FUNCTION_BLOCK fbPPPSZadajnikSR04P
  VAR_INPUT
    sKomunikat : alSTRINGKomunikat;  (* komunikat z systemu zewnętrznego *)
    intTablicaKomunikatowRozmiar : INT;  (* rozmiar tablicy danych wysyłkowych *)
    intModbusOdczytZapisZadanieRozmiar : INT;  (* rozmiar tablicy danych modbusa *)
    xTablicaKomunikatowHold : BOOL;  (* wstrzymanie komunikacji mniej ważnych komunikatów *)
    sIdInstancji : STRING;  (* parametr ID rolety np NS02L*202IBM**** *)
    sIdAplikacji : STRING;  (* parametr ID aplikacji np SO*******ECL*000 *)
    sMnemonik : STRING;  (* mnemonik właściciela - BCB* *)
    sMACAdres : STRING;  (* MAC adres sterownika *)
    sDaneZapasowe : STRING;  (* 6 znaków zapasu *)
    tCzasOpoznieniaRestartu : TIME;  (* czas opóźnienia po którym zaczynają być raportowane wartości *)
    sTypPomieszczenia : STRING;  (* typ pomieszczenia *)
    bAdres : BYTE;
    bKanalEnOcean : BYTE;
    sEnOceanID : STRING(10);
    tMinimalnyCzasRaportowania : TIME;
    tMaksymalnyCzasRaportowania : TIME;
    tCzasTimeoutEnOcean : TIME;
    xAutonomizacja : BOOL;
    xAutonomizacjaSztuczna : BOOL;
    xGlobalnaAutomatycznaKonfiguracja : BOOL;
    tCzestotliwoscAutomatycznejKonfiguracji : TIME;
    rRegulatorTemperaturyKp : REAL;
    rRegulatorTemperaturyTi : REAL;
    rRegulatorTemperaturyDeadZone : REAL;
    rTrybPracyAutonomizacja : REAL;  (* Domyślny tryb pracy *)
    rTemperaturaBazowaAutoAutonomizacja : REAL;  (* Domyślna wartość nastawy temperatury bazowej w trybie automatycznym *)
    rTemperaturaBazowaManAutonomizacja : REAL;  (* Domyślna wartość nastawy temperatury bazowej w trybie manualnym *)
    rSkalaPotencjometruAutonomizacja : REAL;  (* Domyślna skala potencjomentru *)
    rTemperaturaBazowaHMI : REAL := 293.15;  (* Temperatura bazowa z HMI *)
    intTrybPracyHMI : INT := 1;  (* 0 - ręczny; 1 - auto *)
    xPokazPanelHMI : BOOL := TRUE;  (* 0 - widoczny; 1 - niewidoczny *)
  END_VAR
  VAR_IN_OUT
    arModbusOdczytCykliczny : ARRAY[1..5000] OF typModbusOdczytCykliczny;
    arModbusStatusKomunikacji : ARRAY[1..256] OF INT;
    arModbusOdczytZapisZadanie : ARRAY[1..1000] OF typModbusOdczytZapisZadanie;
    intModbusOdczytZapisZadanieZnacznikZapisu : INT;
    arTablicaKomunikatow : alARRAYTablicaKomunikatow;
    intTablicaKomunikatowZnacznikZapisu : INT;
  END_VAR
  VAR_OUTPUT
    rWyjscieRgulatoraTemperatury : REAL;
    rDiagnostykaTemperaturaPomieszczenia : REAL;
    rDiagnostykaTemperaturaNastawiona : REAL;
    rDiagnostykaTemperaturaBazowa : REAL;
    rDiagnostykaKorektaTemperaturyPotencjometru : REAL;
    rDiagnostykaWyjscieRgulatoraTemperatury : REAL;
    intDiagnostykaTrybPracy : INT;
    sDiagnostykaEnOceanIDodczytany : STRING(10);
    wDiagnostykaCzasOdOstatniegoKomunikatu : WORD;
    rTemperaturaPomieszczenia : REAL;
  END_VAR
  VAR CONSTANT
    uintLiczbaRejestrowNaKanal : UINT := 20;
    uintPierwszyRejestr : UINT := 200;
    wEnOceanFunction : WORD := 16;
    wEnOceanType : WORD := 3;
    wEnOceanManufacturer : WORD := 2;
    intDomyslneHarmonogram : INT := enumPPPSHarmonogramy.Komfort;  (* domyślne nastawy po restarcie sterownika *)
    rDomyslneTemperaturaBazowaKomfort : REAL := 293.15;
    rDomyslneTemperaturaBazowaEkonomiczny : REAL := 292.15;
  END_VAR
  VAR
    uintFunctionModbusAdres : UINT;  (* definicja adresów rejestrów modbusowych *)
    uintTypeModbusAdres : UINT;
    uintManufacturerModbusAdres : UINT;
    uintEnOceanIDHiModbusAdres : UINT;
    uintEnOceanIDLoModbusAdres : UINT;
    uintCzasOdOstatniegoKomunikatuModbusAdres : UINT;
    uintPustyRejestr1ModbusAdres : UINT;
    uintStatusUrzadzeniaModbusAdres : UINT;
    uintPustyRejestr2ModbusAdres : UINT;
    uintTemperaturaPomieszczeniaOdczytanaModbusAdres : UINT;
    uintNastawaPotencjometruModbusAdres : UINT;
    xPierwszySkan : BOOL := TRUE;  (* uintLiczbaTelegramowModbusAdres : UINT; zmienne operacyjne *)
    intPetlaPierwszySkan : INT := 1;
    intRozkazTymczasowy : INT;
    arNastawyRegulatoraTemperatury : typConfigPIDController;
    fbRegulatorTemperatury : FbPIDController;
    intBlokadaWykonywaniaRozkazow : INT;
    intBlokadaWykonywaniaRozkazowZaraportowana : INT;
    intTrybPracy : INT;  (* Tryb pracy regulatora. *)
    intTrybPracyZaraportowana : INT;
    xTrybPracyZapisz : BOOL;  (* Trigger zapisu wartości w pamięci urządzenia. *)
    rTrybPracyZapis : REAL;  (* Wartość do zapisania w pamięci urządzenia. *)
    rTemperaturaBazowaAuto : REAL := 293.15;  (* Temperatura bazowa trybu automatycznego. *)
    rTemperaturaBazowaAutoZaraportowana : REAL;
    xTemperaturaBazowaAutoZapisz : BOOL;  (* Trigger zapisu wartości w pamięci urządzenia. *)
    rTemperaturaBazowaAutoZapis : REAL;  (* Wartość do zapisania w pamięci urządzenia. *)
    rTemperaturaBazowaMan : REAL := 293.15;  (* Temperatura bazowa trybu manualnego. *)
    rTemperaturaBazowaManZaraportowana : REAL;
    xTemperaturaBazowaManZapisz : BOOL;  (* Trigger zapisu wartości w pamięci urządzenia. *)
    rTemperaturaBazowaManZapis : REAL;  (* Wartość do zapisania w pamięci urządzenia. *)
    rSkalaPotencjometru : REAL;  (* Skala Potencjometru *)
    rSkalaPotencjometruZaraportowana : REAL;
    xSkalaPotencjometruZapisz : BOOL;  (* Trigger zapisu wartości w pamięci urządzenia. *)
    rSkalaPotencjometruZapis : REAL;  (* Wartość do zapisania w pamięci urządzenia. *)
    fbZadanieGrzania : fbFiltrWartoscAnalogowa;
    rZadanieGrzania : REAL;  (* Zadana grzania *)
    fbZadanieGrzaniaRaport : fbFiltrWartoscAnalogowa;
    rZadanieGrzaniaRaport : REAL;  (* Zadana grzania (raportowana) *)
    rZadanieGrzaniaRaportZaraportowana : REAL;
    rWartoscWejsciowaTemperaturyNastawionej : REAL;
    fbWyslanieKonfiguracji : TON;  (* definicja zmiennych i FB do odczytu wartości z modbusa *)
    xPozwolenieNaAutomatycznaKonfiguracje : BOOL;
    xResetTimerautomatycznejKonfiguracji : BOOL;
    wFunctionEnOceanOdczytana : WORD;
    wTypeEnOceanOdczytana : WORD;
    wManufacturerEnOceanOdczytana : WORD;
    sEnOceanIDodczytany : STRING(10);
    wEnOceanIDHi : WORD;
    wEnOceanIDLo : WORD;
    wEnOceanIDHiZapis : WORD;
    wEnOceanIDLoZapis : WORD;
    wCzasOdOstatniegoKomunikatu : WORD;
    fbTimeoutEnOcean : TON;
    wStatusUrzadzenia : WORD;
    wLiczbaTelegramow : WORD;
    uintLiczbaTelegramow : UINT;
    wPustyRejestr1 : WORD;  (* Rejestry odczytywane dla zgrupowania zapytania rejestrów Modbus *)
    wPustyRejestr2 : WORD;
    wTemperaturaPomieszczeniaOdczytana : WORD;
    fbTemperaturaPomieszczenia : fbFiltrWartoscAnalogowa;
    rTemperaturaPomieszczeniaZaraportowana : REAL;
    wNastawaPotencjometru : WORD;
    rTemperaturaNastawiona : REAL;
    rTemperaturaNastawionaZaraportowana : REAL;
    xPoInicjalizacji : BOOL := FALSE;  (* inicjalizacja *)
    fbInicjalizacyjnyTimer : TON;
    sDane : alSTRINGKomunikat;
    sWyslanyKomunikat : alSTRINGKomunikat;
    sKomunikatPamiec : alSTRINGKomunikat;
    sWyslanyKomunikatDummy : alSTRINGKomunikat;
    intPetla : INT;
    arErrorStan : ARRAY[0..3] OF INT;  (* tablica przechowująca statusy alarmowe *)
    arErrorKlasa : ARRAY[0..3] OF INT;  (* tablica przechowująca klasy danych alarmów *)
    sTempWartoscAtrybutu : STRING;
    rTempWartoscAtrybutu : REAL;
    intTempWartoscAtrybutu : INT;
    xRaport : BOOL;
    uintFunctionAdres : UINT;
    sPlakietkaHMI : STRING;  (* Plakietka pomieszczenia zawierająca numer piętra i pomieszczenia (na potrzeby webvisu) *)
    fnPrzywrocDomyslne : R_TRIG;  (* Przywracanie domyślnych wartości nastaw *)
    fbTaktowanieZapisywaniaModbus : TON;  (* Cykliczne żądanie zapisu danych do urządzenia *)
    xBrakKomunikacjiEnOcean : BOOL;  (* Brak komunikacji z urządzeniem po enOcean *)
    tonBrakKomunikacjiPLC : TON;
    xBrakKomunikacjiPLC : BOOL;
    xBrakKomunikacjiIZE : BOOL;
    rTemperaturaPomieszczeniaPamiec : REAL;  (* Temperatura zapamiętana w celu porównania z aktualną *)
    xBrakZmianyTemperatury : BOOL;  (* Flaga braku zmiany temperatury *)
    fbBrakZmianyTemperaturyTimer : TON;  (* Timer braku zmiany temperatury (24 godziny) *)
    xBladBrakZmianyTemperatury : BOOL;  (* Błąd braku zmiany temperatury *)
    xOsiagniecieTemperaturyZadanej : BOOL := FALSE;  (* Sprawdzanie czy została osiągnęta zadana temperatura *)
    xOsiagniecieTemperaturyZadanejZaraportowana : BOOL := FALSE;
    xFlagaTrybuPracy : BOOL := FALSE;
    rRoznicaTemperaturyZadanejOrazZaraportowanej : REAL;
  END_VAR

            (*			
Autor:					Paweł Kąkol, 2018-08-06, Artur Wyszomirski
Prawa majątkowe: 		Solwena Sp. z o.o., 
Aktualizacje:			
						2018-08-27-PK: dodanie algorytmu nadpisywania konfiguracji (uczenia) anteny
						2018-09-10-PK: dodanie regulatora temperatury oraz obsługi atrybutów potrzebnych do zadajnika z regulatorem, dodanie alarmowania Timeout komunikacji EnOcean
						2018-09-24-AWy: obsługa trybu manualnego i automatycznego
						2018-09-25-PK: dodanie domyślnego przyjmowania 21 st. C po restarcie sterownika, zanim nastąpi Autonomizacja i komunikacja z IZE.
						2018-15-10-AWy: obsługa harmonogramów
						2018-23-10-JB: przygotowanie atrybutów i alarmów do komunikacji z IZE
						2018-12-12-JB: napisanie od nowa obsługi ramek typu C i Q
						2019-02-26-JB: zmiana deadbandów w filtrach analogowych
						2019-04-08-AWy: usunięcie buga braku wysterowania grzejników w trybie manualnym (usunięcie intTrybPracy <> enumPPPSZadajnikTrybPracy.Manualny AND z linii 473)
						2019-05-13-AWy: zmiana wartości umieszczonej w atrybucie STERGRZ. Wartość rZadanieGrzania jest dzielona przez 100 tak, aby zakres STERGRZ mieścił się między 0 a 1.
						2019-05-16-AWy: modyfikacja warunku na raportowanie. Dopisane: AND arModbusStatusKomunikacji[bAdres] = enumModbusStatus.KomunikacjaPrawidlowa AND xPoInicjalizacji 
						2019-05-17-AWy: rozbicie zmiennej rTemperaturaBazowa na rTemperaturaBazowaAuto i rTemperaturaBazowaMan
						2019-05-21-AWy: modyfikacja przepisywania temperatury bazowej z IZE do lokalnej podczas regulacji IZE. 
						2019-06-05-AWy: załadowanie domyślnych trybów pracy i nastaw po przejściu w tryb autonomizacji
						2019-08-05-AWy: dodanie zmiennej sPlakietkaHMI.
						2019-08-14-AWy: zmiana fbPrzywrocDomyslne z przerzutnika RS na R_TRIG.
						2019-09-23-AWy: modyfikacja generowania wartości zmiennej xBrakKomunikacjiPLC
						2019-10-09-AWy: uzależnienie wystąpienia alarmu braku zmiany temperatury od stanu komunikacji 
						2019-10-10-AWy: przywrócenie zmiennej xBrakKomunikacjiEnOcean na potrzeby alarmów i webvisu z I etapu ENGIE
						2019-10-21-AWy: dodanie dodatkowego filtrowania zadanej grzania przy wysyłaniu ramek do IZE
						2019-10-22-AWy: usunięcie uintLiczbaTelegramowModbusAdres z odczytu po Modbusie
						
Opis:					fb służy do komunikacji po Modbus RTU za pośrednictwem bramek (STC65-RS485) EnOcean z zadajnikami FCP0 (SR04P) na budynkach PPP Sopot (ENGIE) 
*)

// Inicjalizacja sterownika
fbInicjalizacyjnyTimer(IN := NOT xPoInicjalizacji , PT := tCzasOpoznieniaRestartu);
IF fbInicjalizacyjnyTimer.Q THEN
	intTrybPracyZaraportowana := intTrybPracy;
	rTemperaturaBazowaAutoZaraportowana := rTemperaturaBazowaAuto;
	rTemperaturaBazowaManZaraportowana := rTemperaturaBazowaMan;
	rSkalaPotencjometruZaraportowana := rSkalaPotencjometru;
	rTemperaturaNastawionaZaraportowana := rTemperaturaNastawiona;
	rTemperaturaPomieszczeniaZaraportowana := rTemperaturaPomieszczenia;
	rZadanieGrzaniaRaportZaraportowana := rZadanieGrzaniaRaport;
	xOsiagniecieTemperaturyZadanej := xOsiagniecieTemperaturyZadanejZaraportowana;
	xPoInicjalizacji := TRUE;
END_IF

// Włącz autonomizację jeśli sterownik jest w stanie inicjalizacji lub nastąpiło wymuszenie autonomizacji
IF NOT xPoInicjalizacji OR xAutonomizacjaSztuczna = TRUE THEN
	xAutonomizacja := TRUE;
END_IF 

// Kontrola komunikacji
tonBrakKomunikacjiPLC(IN := (wCzasOdOstatniegoKomunikatu > 180 OR arModbusStatusKomunikacji[bAdres] <> enumModbusStatus.KomunikacjaPrawidlowa), PT := T#180S);
IF tonBrakKomunikacjiPLC.Q THEN
	xBrakKomunikacjiPLC := TRUE;
ELSE
	xBrakKomunikacjiPLC := FALSE;
END_IF

IF xAutonomizacja THEN
	xBrakKomunikacjiIZE := TRUE;
ELSE
	xBrakKomunikacjiIZE := FALSE;
END_IF

IF xPierwszySkan THEN
	xPierwszySkan := FALSE;
	WHILE arModbusOdczytCykliczny[intPetlaPierwszySkan].bAdresUrzadzenia <> 0 DO
		intPetlaPierwszySkan := intPetlaPierwszySkan + 1;
	END_WHILE
	
	//ustawienie parametrów regulatora temperatury
	arNastawyRegulatoraTemperatury.rKp := rRegulatorTemperaturyKp;
	arNastawyRegulatoraTemperatury.rTn := rRegulatorTemperaturyTi;
	arNastawyRegulatoraTemperatury.rTd := 0.0;
	arNastawyRegulatoraTemperatury.rOutputMax := 100.0;
	arNastawyRegulatoraTemperatury.rOutputMin := 0.0;
	arNastawyRegulatoraTemperatury.xPresetOn := TRUE;
	arNastawyRegulatoraTemperatury.rPresetValueOn := 0.0;
	arNastawyRegulatoraTemperatury.rPresetValueOff := 0.0;
	arNastawyRegulatoraTemperatury.rDeadZone := rRegulatorTemperaturyDeadZone;
	
	//wyznaczenie adresów rejestrów modbusowych
	uintFunctionModbusAdres := uintPierwszyRejestr + (uintLiczbaRejestrowNaKanal * (BYTE_TO_UINT(bKanalEnOcean) - 1));
	uintTypeModbusAdres := uintFunctionModbusAdres + 1;
	uintManufacturerModbusAdres := uintFunctionModbusAdres + 2;
	
	uintEnOceanIDHiModbusAdres := uintFunctionModbusAdres + 3;
	uintEnOceanIDLoModbusAdres := uintFunctionModbusAdres + 4;
	uintCzasOdOstatniegoKomunikatuModbusAdres := uintFunctionModbusAdres + 6;
	uintPustyRejestr1ModbusAdres := uintFunctionModbusAdres + 7;
	uintStatusUrzadzeniaModbusAdres := uintFunctionModbusAdres + 8;
	uintPustyRejestr2ModbusAdres := uintFunctionModbusAdres + 9;
	uintTemperaturaPomieszczeniaOdczytanaModbusAdres := uintFunctionModbusAdres + 10;
	uintNastawaPotencjometruModbusAdres := uintFunctionModbusAdres + 11;
	//uintLiczbaTelegramowModbusAdres := uintFunctionModbusAdres + 19;
	
//deklaracja rejestrow do odczytu
	//rejestry
	arModbusOdczytCykliczny[intPetlaPierwszySkan].bAdresUrzadzenia := bAdres;
	arModbusOdczytCykliczny[intPetlaPierwszySkan].bFunkcja := TO_BYTE(enumModbusKodyFunkcji.OdczytNRejestrow);
	arModbusOdczytCykliczny[intPetlaPierwszySkan].uiAdresRejestru := uintFunctionModbusAdres;
	arModbusOdczytCykliczny[intPetlaPierwszySkan].ltCzestotliwosc := TIME_TO_LTIME(tMaksymalnyCzasRaportowania);
	arModbusOdczytCykliczny[intPetlaPierwszySkan].pZmiennaReferencyjna := ADR(wFunctionEnOceanOdczytana);
	intPetlaPierwszySkan := intPetlaPierwszySkan + 1;
	
	arModbusOdczytCykliczny[intPetlaPierwszySkan].bAdresUrzadzenia := bAdres;
	arModbusOdczytCykliczny[intPetlaPierwszySkan].bFunkcja := TO_BYTE(enumModbusKodyFunkcji.OdczytNRejestrow);
	arModbusOdczytCykliczny[intPetlaPierwszySkan].uiAdresRejestru := uintTypeModbusAdres;
	arModbusOdczytCykliczny[intPetlaPierwszySkan].ltCzestotliwosc := TIME_TO_LTIME(tMaksymalnyCzasRaportowania);
	arModbusOdczytCykliczny[intPetlaPierwszySkan].pZmiennaReferencyjna := ADR(wTypeEnOceanOdczytana);
	intPetlaPierwszySkan := intPetlaPierwszySkan + 1;
	
	arModbusOdczytCykliczny[intPetlaPierwszySkan].bAdresUrzadzenia := bAdres;
	arModbusOdczytCykliczny[intPetlaPierwszySkan].bFunkcja := TO_BYTE(enumModbusKodyFunkcji.OdczytNRejestrow);
	arModbusOdczytCykliczny[intPetlaPierwszySkan].uiAdresRejestru := uintManufacturerModbusAdres;
	arModbusOdczytCykliczny[intPetlaPierwszySkan].ltCzestotliwosc := TIME_TO_LTIME(tMaksymalnyCzasRaportowania);
	arModbusOdczytCykliczny[intPetlaPierwszySkan].pZmiennaReferencyjna := ADR(wManufacturerEnOceanOdczytana);
	intPetlaPierwszySkan := intPetlaPierwszySkan + 1;
	
	arModbusOdczytCykliczny[intPetlaPierwszySkan].bAdresUrzadzenia := bAdres;
	arModbusOdczytCykliczny[intPetlaPierwszySkan].bFunkcja := TO_BYTE(enumModbusKodyFunkcji.OdczytNRejestrow);
	arModbusOdczytCykliczny[intPetlaPierwszySkan].uiAdresRejestru := uintEnOceanIDHiModbusAdres;
	arModbusOdczytCykliczny[intPetlaPierwszySkan].ltCzestotliwosc := TIME_TO_LTIME(tMaksymalnyCzasRaportowania);
	arModbusOdczytCykliczny[intPetlaPierwszySkan].pZmiennaReferencyjna := ADR(wEnOceanIDHi);
	intPetlaPierwszySkan := intPetlaPierwszySkan + 1;
	
	arModbusOdczytCykliczny[intPetlaPierwszySkan].bAdresUrzadzenia := bAdres;
	arModbusOdczytCykliczny[intPetlaPierwszySkan].bFunkcja := TO_BYTE(enumModbusKodyFunkcji.OdczytNRejestrow);
	arModbusOdczytCykliczny[intPetlaPierwszySkan].uiAdresRejestru := uintEnOceanIDLoModbusAdres;
	arModbusOdczytCykliczny[intPetlaPierwszySkan].ltCzestotliwosc := TIME_TO_LTIME(tMaksymalnyCzasRaportowania);
	arModbusOdczytCykliczny[intPetlaPierwszySkan].pZmiennaReferencyjna := ADR(wEnOceanIDLo);
	intPetlaPierwszySkan := intPetlaPierwszySkan + 1;
	
	arModbusOdczytCykliczny[intPetlaPierwszySkan].bAdresUrzadzenia := bAdres;
	arModbusOdczytCykliczny[intPetlaPierwszySkan].bFunkcja := TO_BYTE(enumModbusKodyFunkcji.OdczytNRejestrow);
	arModbusOdczytCykliczny[intPetlaPierwszySkan].uiAdresRejestru := uintCzasOdOstatniegoKomunikatuModbusAdres;
	arModbusOdczytCykliczny[intPetlaPierwszySkan].ltCzestotliwosc := TIME_TO_LTIME(tMinimalnyCzasRaportowania);
	arModbusOdczytCykliczny[intPetlaPierwszySkan].pZmiennaReferencyjna := ADR(wCzasOdOstatniegoKomunikatu);
	intPetlaPierwszySkan := intPetlaPierwszySkan + 1;
	
	arModbusOdczytCykliczny[intPetlaPierwszySkan].bAdresUrzadzenia := bAdres;
	arModbusOdczytCykliczny[intPetlaPierwszySkan].bFunkcja := TO_BYTE(enumModbusKodyFunkcji.OdczytNRejestrow);
	arModbusOdczytCykliczny[intPetlaPierwszySkan].uiAdresRejestru := uintPustyRejestr1ModbusAdres;
	arModbusOdczytCykliczny[intPetlaPierwszySkan].ltCzestotliwosc := TIME_TO_LTIME(tMinimalnyCzasRaportowania);
	arModbusOdczytCykliczny[intPetlaPierwszySkan].pZmiennaReferencyjna := ADR(wPustyRejestr1);
	intPetlaPierwszySkan := intPetlaPierwszySkan + 1;
	
	arModbusOdczytCykliczny[intPetlaPierwszySkan].bAdresUrzadzenia := bAdres;
	arModbusOdczytCykliczny[intPetlaPierwszySkan].bFunkcja := TO_BYTE(enumModbusKodyFunkcji.OdczytNRejestrow);
	arModbusOdczytCykliczny[intPetlaPierwszySkan].uiAdresRejestru := uintStatusUrzadzeniaModbusAdres;
	arModbusOdczytCykliczny[intPetlaPierwszySkan].ltCzestotliwosc := TIME_TO_LTIME(tMinimalnyCzasRaportowania);
	arModbusOdczytCykliczny[intPetlaPierwszySkan].pZmiennaReferencyjna := ADR(wStatusUrzadzenia);
	intPetlaPierwszySkan := intPetlaPierwszySkan + 1;
	
	arModbusOdczytCykliczny[intPetlaPierwszySkan].bAdresUrzadzenia := bAdres;
	arModbusOdczytCykliczny[intPetlaPierwszySkan].bFunkcja := TO_BYTE(enumModbusKodyFunkcji.OdczytNRejestrow);
	arModbusOdczytCykliczny[intPetlaPierwszySkan].uiAdresRejestru := uintPustyRejestr2ModbusAdres;
	arModbusOdczytCykliczny[intPetlaPierwszySkan].ltCzestotliwosc := TIME_TO_LTIME(tMinimalnyCzasRaportowania);
	arModbusOdczytCykliczny[intPetlaPierwszySkan].pZmiennaReferencyjna := ADR(wPustyRejestr2);
	intPetlaPierwszySkan := intPetlaPierwszySkan + 1;
	
	arModbusOdczytCykliczny[intPetlaPierwszySkan].bAdresUrzadzenia := bAdres;
	arModbusOdczytCykliczny[intPetlaPierwszySkan].bFunkcja := TO_BYTE(enumModbusKodyFunkcji.OdczytNRejestrow);
	arModbusOdczytCykliczny[intPetlaPierwszySkan].uiAdresRejestru := uintTemperaturaPomieszczeniaOdczytanaModbusAdres;
	arModbusOdczytCykliczny[intPetlaPierwszySkan].ltCzestotliwosc := TIME_TO_LTIME(tMinimalnyCzasRaportowania);
	arModbusOdczytCykliczny[intPetlaPierwszySkan].pZmiennaReferencyjna := ADR(wTemperaturaPomieszczeniaOdczytana);
	intPetlaPierwszySkan := intPetlaPierwszySkan + 1;	
	
	arModbusOdczytCykliczny[intPetlaPierwszySkan].bAdresUrzadzenia := bAdres;
	arModbusOdczytCykliczny[intPetlaPierwszySkan].bFunkcja := TO_BYTE(enumModbusKodyFunkcji.OdczytNRejestrow);
	arModbusOdczytCykliczny[intPetlaPierwszySkan].uiAdresRejestru := uintNastawaPotencjometruModbusAdres;
	arModbusOdczytCykliczny[intPetlaPierwszySkan].ltCzestotliwosc := TIME_TO_LTIME(tMinimalnyCzasRaportowania);
	arModbusOdczytCykliczny[intPetlaPierwszySkan].pZmiennaReferencyjna := ADR(wNastawaPotencjometru);
	intPetlaPierwszySkan := intPetlaPierwszySkan + 1;
(*	
	arModbusOdczytCykliczny[intPetlaPierwszySkan].bAdresUrzadzenia := bAdres;
	arModbusOdczytCykliczny[intPetlaPierwszySkan].bFunkcja := TO_BYTE(enumModbusKodyFunkcji.OdczytNRejestrow);
	arModbusOdczytCykliczny[intPetlaPierwszySkan].uiAdresRejestru := uintLiczbaTelegramowModbusAdres;
	arModbusOdczytCykliczny[intPetlaPierwszySkan].ltCzestotliwosc := TIME_TO_LTIME(tMinimalnyCzasRaportowania);
	arModbusOdczytCykliczny[intPetlaPierwszySkan].pZmiennaReferencyjna := ADR(wLiczbaTelegramow);
	intPetlaPierwszySkan := intPetlaPierwszySkan + 1;
*)	
(*	//przyjęcie nastaw domyślnych do momentu uzyskania nastaw z IZE lub przejścia w autonomizację
	IF intDomyslneHarmonogram = enumPPPSHarmonogramy.Ekonomiczny THEN
		rTemperaturaBazowaAuto := rDomyslneTemperaturaBazowaEkonomiczny;
	ELSE
		rTemperaturaBazowaAuto := rDomyslneTemperaturaBazowaKomfort;													
	END_IF
	intTrybPracy := enumPPPSZadajnikTrybPracy.Automatyczny;
	rSkalaPotencjometru := rSkalaPotencjometruAutonomizacja;	*)
END_IF

// Obsługa komunikatu przychodzacego z IZE
IF 	sKomunikat <> sKomunikatPamiec AND xPoInicjalizacji THEN
	sKomunikatPamiec := sKomunikat;
	IF fnIDOdbiorcyMatch(sKomunikat , sIdInstancji) THEN
		sDane := '';
		// Rozkaz typu C
		IF fnKomunikatTyp(sKomunikat) = 'C' AND NOT xAutonomizacja THEN
			// Blokada wykonywania rozkazów
			IF fnKomunikatDaneSzukajWartosci(sKomunikat,'BLOK=') = '0' THEN
				IF intBlokadaWykonywaniaRozkazow = 1 THEN
					intBlokadaWykonywaniaRozkazow := 0;
					xRaport := TRUE;
					ELSE	
					IF sDane <> '' THEN
					sDane := CONCAT(sDane , ';');
					END_IF
					sDane := CONCAT(sDane , 'BLOK=0');
				END_IF
			END_IF
			IF fnKomunikatDaneSzukajWartosci(sKomunikat,'BLOK=') = '1' THEN
				IF intBlokadaWykonywaniaRozkazow = 0 THEN
					intBlokadaWykonywaniaRozkazow := 1;
					xRaport := TRUE;
					ELSE
					IF sDane <> '' THEN
					sDane := CONCAT(sDane , ';');
					END_IF					
					sDane := CONCAT(sDane , 'BLOK=1');
				END_IF
			END_IF		

			IF intBlokadaWykonywaniaRozkazow = 0 THEN
				// Tryby pracy 
				fnKomunikatDaneZnajdzPorownajZapisz(sKomunikat := sKomunikat,
					sAtrybut := 'TRYB=',
					rAtrybutWartosc := rTrybPracyZapis,
					sDane := sDane,
					xAtrybutZapisz => xTrybPracyZapisz);	
				// Temperatura bazowa w trybie automatycznym
				fnKomunikatDaneZnajdzPorownajZapisz(sKomunikat := sKomunikat,
					sAtrybut := 'TEMPBAZAUTO=',
					rAtrybutWartosc := rTemperaturaBazowaAutoZapis,
					sDane := sDane,
					xAtrybutZapisz => xTemperaturaBazowaAutoZapisz);	
				// Temperatura bazowa w trybie manualnym
				fnKomunikatDaneZnajdzPorownajZapisz(sKomunikat := sKomunikat,
					sAtrybut := 'TEMPBAZMAN=',
					rAtrybutWartosc := rTemperaturaBazowaManZapis,
					sDane := sDane,
					xAtrybutZapisz => xTemperaturaBazowaManZapisz);
				// Skala potencjometru
				fnKomunikatDaneZnajdzPorownajZapisz(sKomunikat := sKomunikat,
					sAtrybut := 'SKALAPOT=',
					rAtrybutWartosc := rSkalaPotencjometruZapis,
					sDane := sDane,
					xAtrybutZapisz => xSkalaPotencjometruZapisz);
			END_IF
		END_IF	

		// Zapytanie typu Q
		IF fnKomunikatTyp(sKomunikat) = 'Q' AND arModbusStatusKomunikacji[bAdres] = enumModbusStatus.KomunikacjaPrawidlowa THEN
			IF fnKomunikatDaneSzukajWartosci(sKomunikat , 'BLOK=') = '?' OR fnKomunikatDaneSzukajWartosci(sKomunikat , 'ALL=') = '?' THEN
				fnKomunikatDaneDodaj(sDane := sDane , sAtrybut := 'BLOK=' , sWartosc := INT_TO_STRING(intBlokadaWykonywaniaRozkazow));	
			END_IF
			IF fnKomunikatDaneSzukajWartosci(sKomunikat , 'TRYB=') = '?' OR fnKomunikatDaneSzukajWartosci(sKomunikat , 'ALL=') = '?' THEN
				fnKomunikatDaneDodaj(sDane := sDane , sAtrybut := 'TRYB=' , sWartosc := INT_TO_STRING(intTrybPracy));	
			END_IF
			IF (fnKomunikatDaneSzukajWartosci(sKomunikat , 'TEMPBAZMAN=') = '?' OR fnKomunikatDaneSzukajWartosci(sKomunikat , 'ALL=') = '?') THEN
				fnKomunikatDaneDodaj(sDane := sDane , sAtrybut := 'TEMPBAZMAN=' , sWartosc := REAL_TO_STRING(rTemperaturaBazowaMan));	
			END_IF
			IF (fnKomunikatDaneSzukajWartosci(sKomunikat , 'TEMPBAZAUTO=') = '?' OR fnKomunikatDaneSzukajWartosci(sKomunikat , 'ALL=') = '?') THEN
				fnKomunikatDaneDodaj(sDane := sDane , sAtrybut := 'TEMPBAZAUTO=' , sWartosc := REAL_TO_STRING(rTemperaturaBazowaAuto));	
			END_IF
			IF fnKomunikatDaneSzukajWartosci(sKomunikat , 'SKALAPOT=') = '?' OR fnKomunikatDaneSzukajWartosci(sKomunikat , 'ALL=') = '?' THEN
				fnKomunikatDaneDodaj(sDane := sDane , sAtrybut := 'SKALAPOT=' , sWartosc := REAL_TO_STRING(rSkalaPotencjometru));	
			END_IF
			IF fnKomunikatDaneSzukajWartosci(sKomunikat , 'TEMP=') = '?' OR fnKomunikatDaneSzukajWartosci(sKomunikat , 'ALL=') = '?' THEN
				fnKomunikatDaneDodaj(sDane := sDane , sAtrybut := 'TEMP=' , sWartosc := REAL_TO_STRING(rTemperaturaPomieszczenia));	
			END_IF
			IF fnKomunikatDaneSzukajWartosci(sKomunikat , 'STERGRZ=') = '?' OR fnKomunikatDaneSzukajWartosci(sKomunikat , 'ALL=') = '?' THEN
				fnKomunikatDaneDodaj(sDane := sDane , sAtrybut := 'STERGRZ=' , sWartosc := REAL_TO_STRING(rZadanieGrzaniaRaport / 100));	
			END_IF
			IF fnKomunikatDaneSzukajWartosci(sKomunikat , 'TEMPNAS=') = '?' OR fnKomunikatDaneSzukajWartosci(sKomunikat , 'ALL=') = '?' THEN
				fnKomunikatDaneDodaj(sDane := sDane , sAtrybut := 'TEMPNAS=' , sWartosc := REAL_TO_STRING(rTemperaturaNastawiona));	
			END_IF
			IF fnKomunikatDaneSzukajWartosci(sKomunikat , 'DOGRZ=') = '?' OR fnKomunikatDaneSzukajWartosci(sKomunikat , 'ALL=') = '?' THEN
				fnKomunikatDaneDodaj(sDane := sDane , sAtrybut := 'DOGRZ=' , sWartosc := INT_TO_STRING(BOOL_TO_INT(xOsiagniecieTemperaturyZadanej)));	
			END_IF
			//pytanie o stany alarmów
			IF fnKomunikatDaneSzukajWartosci(sKomunikat , 'ALARM=') = '?' OR fnKomunikatDaneSzukajWartosci(sKomunikat , 'ALL=') = '?' THEN
				FOR intPetla := 1 TO 4 BY 1 DO
					//raportowanie typu E (stanów alarmów) na zapytanie typu Q
					IF arErrorStan[intPetla] <> enumAlarmWartosc.StanNieznany THEN
						fnZapiszKomunikat(	sCalyKomunikat := '' ,
											sTypKomunikatu := 'E' ,
											sMnemonik := sMnemonik ,
											sMACAdres := sMACAdres ,
											sIDNadawcy := sIdInstancji ,
											sIDOdbiorcy := sIdAplikacji ,
											sDaneZapasowe := sDaneZapasowe ,
											sDane := fnKomunikatDaneErrorRetry(xAktywny := arErrorStan[intPetla] = enumAlarmWartosc.StanAlarmowy , intKlasa := arErrorKlasa[intPetla] , intNumer := intPetla),
											arTablicaKomunikatow := arTablicaKomunikatow ,
											intTablicaKomunikatowZnacznikZapisu := intTablicaKomunikatowZnacznikZapisu ,
											intTablicaKomunikatowRozmiar := intTablicaKomunikatowRozmiar ,
											sWyslanyKomunikat := sWyslanyKomunikatDummy);
					END_IF
				END_FOR
			END_IF
		END_IF
		
		// Raportowanie typu A
		IF sDane <> '' THEN
			fnZapiszKomunikat(	sCalyKomunikat := '' ,
								sTypKomunikatu := 'A' ,
								sMnemonik := sMnemonik ,
								sMACAdres := sMACAdres ,
								sIDNadawcy := sIdInstancji ,
								sIDOdbiorcy := sIdAplikacji ,
								sDaneZapasowe := sDaneZapasowe ,
								sDane := sDane ,
								arTablicaKomunikatow := arTablicaKomunikatow ,
								intTablicaKomunikatowZnacznikZapisu := intTablicaKomunikatowZnacznikZapisu ,
								intTablicaKomunikatowRozmiar := intTablicaKomunikatowRozmiar ,
								sWyslanyKomunikat := sWyslanyKomunikatDummy);
		END_IF
	END_IF
END_IF

// Przywrócenie wartości domyślnych nastaw krzywej grzewczej i trybów pracy w przypadku restartu sterownika lub przejścia w stan autonomizacji (brak komunikacji z IZE)
fnPrzywrocDomyslne(CLK := xAutonomizacja);
IF fnPrzywrocDomyslne.Q THEN	
	IF intTrybPracy <> REAL_TO_INT(rTrybPracyAutonomizacja) THEN
		rTrybPracyZapis := rTrybPracyAutonomizacja;
		xTrybPracyZapisz := TRUE;
	END_IF
	IF rTemperaturaBazowaAuto <> rTemperaturaBazowaAutoAutonomizacja THEN
		rTemperaturaBazowaAutoZapis := rTemperaturaBazowaAutoAutonomizacja + 273.15;
		xTemperaturaBazowaAutoZapisz := TRUE;
	END_IF
	IF rTemperaturaBazowaMan <> rTemperaturaBazowaManAutonomizacja THEN
		rTemperaturaBazowaManZapis := rTemperaturaBazowaManAutonomizacja;
		xTemperaturaBazowaManZapisz := TRUE;
	END_IF
	IF rSkalaPotencjometru <> rSkalaPotencjometruAutonomizacja THEN
		rSkalaPotencjometruZapis := rSkalaPotencjometruAutonomizacja;
		xSkalaPotencjometruZapisz := TRUE;
	END_IF
END_IF	

// Zapisanie nastaw domyślnych lub otrzymanych w ramce C
IF xTrybPracyZapisz THEN
	intTrybPracy := REAL_TO_INT(rTrybPracyZapis);
	intTrybPracyHMI := REAL_TO_INT(rTrybPracyZapis);
	xTrybPracyZapisz := FALSE;
END_IF
IF xTemperaturaBazowaAutoZapisz THEN
	rTemperaturaBazowaAuto := rTemperaturaBazowaAutoZapis;
	xTemperaturaBazowaAutoZapisz := FALSE;
END_IF
IF xTemperaturaBazowaManZapisz THEN
	rTemperaturaBazowaMan := rTemperaturaBazowaManZapis;
	xTemperaturaBazowaManZapisz := FALSE;
END_IF
IF xSkalaPotencjometruZapisz THEN
	rSkalaPotencjometru := rSkalaPotencjometruZapis;
	xSkalaPotencjometruZapisz := FALSE;
END_IF

// Tryby pracy
IF xAutonomizacja THEN	// W trybie automonizacji pobieraj tryb pracy i temperaturę bazową z panelu WebVisu
	IF intTrybPracyHMI = enumPPPSZadajnikTrybPracy.Manualny THEN	
		intTrybPracy := enumPPPSZadajnikTrybPracy.Manualny;
		rTemperaturaBazowaMan := rTemperaturaBazowaHMI + 273.15;
	ELSE
		intTrybPracy := enumPPPSZadajnikTrybPracy.Automatyczny;
		rTemperaturaBazowaAuto := rTemperaturaBazowaAutoAutonomizacja + 273.15;
	END_IF
ELSE // W trybie sterowania z IZE pobieraj tryb pracy i temperaturę bazową z panelu WebVisu
	IF intTrybPracy = enumPPPSZadajnikTrybPracy.Manualny THEN
		intTrybPracyHMI := enumPPPSZadajnikTrybPracy.Manualny;
		rTemperaturaBazowaHMI := rTemperaturaBazowaMan - 273.15;
	ELSE
		intTrybPracyHMI := enumPPPSZadajnikTrybPracy.Automatyczny;
		rTemperaturaBazowaHMI := rTemperaturaBazowaAuto - 273.15;
	END_IF	
END_IF
						 
IF intTrybPracy = enumPPPSZadajnikTrybPracy.Manualny THEN 	
	rTemperaturaNastawiona := rTemperaturaBazowaMan; // W trybie manualnym nie uwzględniaj nastawy potencjometru na zadajniku
ELSE
	rTemperaturaNastawiona := ((WORD_TO_REAL(wNastawaPotencjometru) - 127.0) * rSkalaPotencjometru / 127.0) + rTemperaturaBazowaAuto; // W trybie automatycznym uwzględnij nastawę Potencjometru
END_IF

//Autokonfiguracja bramki EnOcean
sEnOceanIDodczytany := CONCAT(CONCAT(fnKonwersjaDEC_BYTE_TO_HEX_STRING(INT_TO_BYTE(WORD_TO_INT(wEnOceanIDHi / 256))), fnKonwersjaDEC_BYTE_TO_HEX_STRING(WORD_TO_BYTE(wEnOceanIDHi))), CONCAT(fnKonwersjaDEC_BYTE_TO_HEX_STRING(INT_TO_BYTE(WORD_TO_INT(wEnOceanIDLo / 256))), fnKonwersjaDEC_BYTE_TO_HEX_STRING(WORD_TO_BYTE(wEnOceanIDLo))));

fbWyslanieKonfiguracji(IN := ((xPozwolenieNaAutomatycznaKonfiguracje OR xGlobalnaAutomatycznaKonfiguracja) AND NOT xResetTimerautomatycznejKonfiguracji) , PT := tCzestotliwoscAutomatycznejKonfiguracji);
xResetTimerautomatycznejKonfiguracji := FALSE;

IF((xPozwolenieNaAutomatycznaKonfiguracje OR xGlobalnaAutomatycznaKonfiguracja) AND fbWyslanieKonfiguracji.Q) THEN
	//EnOcean ID urządzenia
	IF sEnOceanID <> sEnOceanIDodczytany THEN
		wEnOceanIDHiZapis := BYTE_TO_WORD(fnKonwersjaHEX_STRING_TO_DEC_BYTE(LEFT(sEnOceanID, 2))) * 256 + BYTE_TO_WORD(fnKonwersjaHEX_STRING_TO_DEC_BYTE(LEFT(RIGHT(sEnOceanID, 6), 2)));
		fnModbusZapisRejestru(	bAdresUrzadzenia := bAdres,
								bFunkcja := INT_TO_BYTE(enumModbusKodyFunkcji.ZapisRejestru),										
								uiAdresRejestru := uintEnOceanIDHiModbusAdres,
								pZmiennaReferencyjna := 0,
								wWartoscDoZapisania := wEnOceanIDHiZapis,
								intModbusOdczytZapisZadanieRozmiar := intModbusOdczytZapisZadanieRozmiar,
								arModbusOdczytZapisZadanie := arModbusOdczytZapisZadanie,
								intModbusOdczytZapisZadanieZnacznikZapisu := intModbusOdczytZapisZadanieZnacznikZapisu);
		wEnOceanIDLoZapis := BYTE_TO_WORD(fnKonwersjaHEX_STRING_TO_DEC_BYTE(LEFT(RIGHT(sEnOceanID, 4), 2))) * 256 + BYTE_TO_WORD(fnKonwersjaHEX_STRING_TO_DEC_BYTE(RIGHT(sEnOceanID, 2)));
		fnModbusZapisRejestru(	bAdresUrzadzenia := bAdres,
								bFunkcja := INT_TO_BYTE(enumModbusKodyFunkcji.ZapisRejestru),										
								uiAdresRejestru := uintEnOceanIDLoModbusAdres,
								pZmiennaReferencyjna := 0,
								wWartoscDoZapisania := wEnOceanIDLoZapis,
								intModbusOdczytZapisZadanieRozmiar := intModbusOdczytZapisZadanieRozmiar,
								arModbusOdczytZapisZadanie := arModbusOdczytZapisZadanie,
								intModbusOdczytZapisZadanieZnacznikZapisu := intModbusOdczytZapisZadanieZnacznikZapisu);
	END_IF
	//stałe wartości dla danego typu urządzeń
	IF wFunctionEnOceanOdczytana <> wEnOceanFunction THEN
		fnModbusZapisRejestru(	bAdresUrzadzenia := bAdres,
								bFunkcja := INT_TO_BYTE(enumModbusKodyFunkcji.ZapisRejestru),										
								uiAdresRejestru := uintFunctionModbusAdres,
								pZmiennaReferencyjna := 0,
								wWartoscDoZapisania := wEnOceanFunction,
								intModbusOdczytZapisZadanieRozmiar := intModbusOdczytZapisZadanieRozmiar,
								arModbusOdczytZapisZadanie := arModbusOdczytZapisZadanie,
								intModbusOdczytZapisZadanieZnacznikZapisu := intModbusOdczytZapisZadanieZnacznikZapisu);
	END_IF
	IF wTypeEnOceanOdczytana <> wEnOceanType THEN
		fnModbusZapisRejestru(	bAdresUrzadzenia := bAdres,
								bFunkcja := INT_TO_BYTE(enumModbusKodyFunkcji.ZapisRejestru),										
								uiAdresRejestru := uintTypeModbusAdres,
								pZmiennaReferencyjna := 0,
								wWartoscDoZapisania := wEnOceanType,
								intModbusOdczytZapisZadanieRozmiar := intModbusOdczytZapisZadanieRozmiar,
								arModbusOdczytZapisZadanie := arModbusOdczytZapisZadanie,
								intModbusOdczytZapisZadanieZnacznikZapisu := intModbusOdczytZapisZadanieZnacznikZapisu);
	END_IF
	IF wManufacturerEnOceanOdczytana <> wEnOceanManufacturer THEN
		fnModbusZapisRejestru(	bAdresUrzadzenia := bAdres,
								bFunkcja := INT_TO_BYTE(enumModbusKodyFunkcji.ZapisRejestru),										
								uiAdresRejestru := uintManufacturerModbusAdres,
								pZmiennaReferencyjna := 0,
								wWartoscDoZapisania := wEnOceanManufacturer,
								intModbusOdczytZapisZadanieRozmiar := intModbusOdczytZapisZadanieRozmiar,
								arModbusOdczytZapisZadanie := arModbusOdczytZapisZadanie,
								intModbusOdczytZapisZadanieZnacznikZapisu := intModbusOdczytZapisZadanieZnacznikZapisu);
	END_IF
	xResetTimerautomatycznejKonfiguracji := TRUE;
END_IF

//sprawdzanie Timeout komunikacji
fbTimeoutEnOcean(IN := ((wCzasOdOstatniegoKomunikatu > 120) AND arModbusStatusKomunikacji[bAdres] = enumModbusStatus.KomunikacjaPrawidlowa) , PT := tCzasTimeoutEnOcean);	
							
fbTemperaturaPomieszczenia(	rWartoscWejsciowa := WORD_TO_REAL(wTemperaturaPomieszczeniaOdczytana),
							rDeadband := 0.1,
							tCzasMinimalny := tMinimalnyCzasRaportowania,
							tCzasMaksymalny := tMaksymalnyCzasRaportowania,
							rWynikMnoznik := (-40.0 / 255.0),
							rWynikOffset := 273.15 + 40.0,
							rWartoscWejsciowaZaraportowana := rTemperaturaPomieszczeniaZaraportowana,
							rWartoscWyjsciowa => rTemperaturaPomieszczenia);

//regulator PI
fbRegulatorTemperatury( xEnable := TRUE,
	rReferenceValue := rTemperaturaNastawiona,
	rActualValue := rTemperaturaPomieszczenia,
	typConfigParameters := arNastawyRegulatoraTemperatury,
	rY => rWyjscieRgulatoraTemperatury);

fbZadanieGrzania(rWartoscWejsciowa := rWyjscieRgulatoraTemperatury,
	rDeadband := 0.25,
	tCzasMinimalny := tMinimalnyCzasRaportowania,
	tCzasMaksymalny := tMaksymalnyCzasRaportowania,
	rWynikMnoznik := 1,
	rWynikOffset := 0.0,
	rWartoscWejsciowaZaraportowana := rZadanieGrzania,
	rWartoscWyjsciowa => rZadanieGrzania);		
	
// Raportowanie zadanej grzania
fbZadanieGrzaniaRaport(rWartoscWejsciowa := rZadanieGrzania,
	rDeadband := 10,
	tCzasMinimalny := tMinimalnyCzasRaportowania,
	tCzasMaksymalny := tMaksymalnyCzasRaportowania,
	rWynikMnoznik := 1,
	rWynikOffset := 0.0,
	rWartoscWejsciowaZaraportowana := rZadanieGrzaniaRaportZaraportowana,
	rWartoscWyjsciowa => rZadanieGrzaniaRaport);		
	
// Nowy filtr "antypyćkowy"
IF rZadanieGrzania < 0.25 THEN
	rZadanieGrzania := 0;
	rZadanieGrzaniaRaport := 0;
ELSIF rZadanieGrzania > 99.75 THEN
	rZadanieGrzania := 100;
	rZadanieGrzaniaRaport := 100;	
END_IF
(*
// FILTR ANTY_PYĆKOWY
rRoznicaTemperaturyZadanejOrazZaraportowanej := rZadanieGrzania - rZadanieGrzaniaZaraportowana;
IF rRoznicaTemperaturyZadanejOrazZaraportowanej < 0.25 AND rRoznicaTemperaturyZadanejOrazZaraportowanej > 0 AND rZadanieGrzania < 1.0 THEN
	rZadanieGrzania := rZadanieGrzaniaZaraportowana;
END_IF	

IF rRoznicaTemperaturyZadanejOrazZaraportowanej > - 0.25 AND rRoznicaTemperaturyZadanejOrazZaraportowanej < 0 AND rZadanieGrzania > 99.0 THEN
	rZadanieGrzania := rZadanieGrzaniaZaraportowana;
END_IF	
	*)		
///////Diagnostyka na czas uruchomień////////
	rDiagnostykaTemperaturaPomieszczenia := rTemperaturaPomieszczenia;
	rDiagnostykaTemperaturaNastawiona := rTemperaturaNastawiona;
	rDiagnostykaTemperaturaBazowa := rTemperaturaBazowaAuto;
	rDiagnostykaKorektaTemperaturyPotencjometru := (WORD_TO_REAL(wNastawaPotencjometru) - 127.0) * rSkalaPotencjometru / 127.0;
	rDiagnostykaWyjscieRgulatoraTemperatury := rWyjscieRgulatoraTemperatury;
	intDiagnostykaTrybPracy := intTrybPracy;
	sDiagnostykaEnOceanIDodczytany := sEnOceanIDodczytany;
	wDiagnostykaCzasOdOstatniegoKomunikatu := wCzasOdOstatniegoKomunikatu;
//////////////////////////////////////////////		
IF (intBlokadaWykonywaniaRozkazow <> intBlokadaWykonywaniaRozkazowZaraportowana OR intTrybPracy <> intTrybPracyZaraportowana OR rTemperaturaBazowaAuto <> rTemperaturaBazowaAutoZaraportowana OR 
	rSkalaPotencjometru <> rSkalaPotencjometruZaraportowana OR rTemperaturaNastawiona <> rTemperaturaNastawionaZaraportowana OR rTemperaturaPomieszczenia <> rTemperaturaPomieszczeniaZaraportowana OR 
	rZadanieGrzaniaRaport <> rZadanieGrzaniaRaportZaraportowana OR xOsiagniecieTemperaturyZadanej <> xOsiagniecieTemperaturyZadanejZaraportowana OR rTemperaturaBazowaMan <> rTemperaturaBazowaManZaraportowana) AND 
	arModbusStatusKomunikacji[bAdres] = enumModbusStatus.KomunikacjaPrawidlowa AND xPoInicjalizacji THEN
	xRaport := TRUE;
END_IF

IF xRaport THEN
	sDane := '';
	xRaport := FALSE;
	IF intBlokadaWykonywaniaRozkazow <> intBlokadaWykonywaniaRozkazowZaraportowana THEN
		intBlokadaWykonywaniaRozkazowZaraportowana := intBlokadaWykonywaniaRozkazow;
		fnKomunikatDaneDodaj(sDane := sDane , sAtrybut := 'BLOK=' , sWartosc := INT_TO_STRING(intBlokadaWykonywaniaRozkazow));	
	END_IF
	IF intTrybPracy <> intTrybPracyZaraportowana THEN
		intTrybPracyZaraportowana := intTrybPracy;
		fnKomunikatDaneDodaj(sDane := sDane , sAtrybut := 'TRYB=' , sWartosc := INT_TO_STRING(intTrybPracy));	
	END_IF
	IF (rTemperaturaBazowaMan <> rTemperaturaBazowaManZaraportowana) THEN
		rTemperaturaBazowaManZaraportowana := rTemperaturaBazowaMan;
		fnKomunikatDaneDodaj(sDane := sDane , sAtrybut := 'TEMPBAZMAN=' , sWartosc := REAL_TO_STRING(rTemperaturaBazowaMan));	
	END_IF
	IF (rTemperaturaBazowaAuto <> rTemperaturaBazowaAutoZaraportowana) THEN
		rTemperaturaBazowaAutoZaraportowana := rTemperaturaBazowaAuto;
		fnKomunikatDaneDodaj(sDane := sDane , sAtrybut := 'TEMPBAZAUTO=' , sWartosc := REAL_TO_STRING(rTemperaturaBazowaAuto));	
	END_IF
	IF rSkalaPotencjometru <> rSkalaPotencjometruZaraportowana THEN
		rSkalaPotencjometruZaraportowana := rSkalaPotencjometru;
		fnKomunikatDaneDodaj(sDane := sDane , sAtrybut := 'SKALAPOT=' , sWartosc := REAL_TO_STRING(rSkalaPotencjometru));	
	END_IF
	IF rTemperaturaNastawiona <> rTemperaturaNastawionaZaraportowana THEN
		rTemperaturaNastawionaZaraportowana := rTemperaturaNastawiona;
		fnKomunikatDaneDodaj(sDane := sDane , sAtrybut := 'TEMPNAS=' , sWartosc := REAL_TO_STRING(rTemperaturaNastawiona));	
	END_IF
	IF rTemperaturaPomieszczenia <> rTemperaturaPomieszczeniaZaraportowana THEN
		rTemperaturaPomieszczeniaZaraportowana := rTemperaturaPomieszczenia;
		fnKomunikatDaneDodaj(sDane := sDane , sAtrybut := 'TEMP=' , sWartosc := REAL_TO_STRING(rTemperaturaPomieszczenia));	
	END_IF
	IF rZadanieGrzaniaRaport <> rZadanieGrzaniaRaportZaraportowana THEN
		rZadanieGrzaniaRaportZaraportowana := rZadanieGrzaniaRaport;	
		fnKomunikatDaneDodaj(sDane := sDane , sAtrybut := 'STERGRZ=' , sWartosc := REAL_TO_STRING(rZadanieGrzaniaRaport / 100));	
	END_IF
	IF xOsiagniecieTemperaturyZadanej <> xOsiagniecieTemperaturyZadanejZaraportowana THEN
		xOsiagniecieTemperaturyZadanejZaraportowana := xOsiagniecieTemperaturyZadanej;
		fnKomunikatDaneDodaj(sDane := sDane , sAtrybut := 'DOGRZ=' , sWartosc := INT_TO_STRING(BOOL_TO_INT(xOsiagniecieTemperaturyZadanej)));	
	END_IF
	
(*	IF rTemperaturaPomieszczeniaMIN <> rTemperaturaPomieszczeniaMINZaraportowana OR rTemperaturaPomieszczeniaMAX <> rTemperaturaPomieszczeniaMAXZaraportowana THEN
		
		fnKomunikatDaneDodaj(sDane := sDane , sAtrybut := 'TEMPPOC=' , sWartosc := REAL_TO_STRING(rTemperaturaPomieszczeniaPOCZATKOWA));
		rTemperaturaPomieszczeniaPOCZATKOWA := rTemperaturaPomieszczenia;
		
		rTemperaturaPomieszczeniaKONCOWA := rTemperaturaPomieszczenia;
		fnKomunikatDaneDodaj(sDane := sDane , sAtrybut := 'TEMPKON=' , sWartosc := REAL_TO_STRING(rTemperaturaPomieszczeniaKONCOWA));
		
		rTemperaturaPomieszczeniaMINZaraportowana := rTemperaturaPomieszczeniaMIN;
		fnKomunikatDaneDodaj(sDane := sDane , sAtrybut := 'TEMPMIN=' , sWartosc := REAL_TO_STRING(rTemperaturaPomieszczeniaMIN));
		rZmiennaProcesowaMinimumTemperatury := 500.0;
		
		rTemperaturaPomieszczeniaMAXZaraportowana := rTemperaturaPomieszczeniaMAX;
		fnKomunikatDaneDodaj(sDane := sDane , sAtrybut := 'TEMPMAX=' , sWartosc := REAL_TO_STRING(rTemperaturaPomieszczeniaMAX));
		rZmiennaProcesowaMaximumTemperatury := -1.0;
		
		fnKomunikatDaneDodaj(sDane := sDane , sAtrybut := 'TEMPSRE=' , sWartosc := REAL_TO_STRING(rTemperaturaPomieszczeniaSREDNIA));
		rTemperaturaPomieszczeniaSREDNIA := 0.0;
		
		fnKomunikatDaneDodaj(sDane := sDane , sAtrybut := 'TEMPMED=' , sWartosc := REAL_TO_STRING(rTemperaturaPomieszczeniaMEDIANA));
		rTemperaturaPomieszczeniaMEDIANA := -1.0;
	END_IF
*)

	IF sDane <> '' AND xPoInicjalizacji THEN
		fnZapiszKomunikat(	sCalyKomunikat := '' ,
							sTypKomunikatu := 'M' ,
							sMnemonik := sMnemonik ,
							sMACAdres := sMACAdres ,
							sIDNadawcy := sIdInstancji ,
							sIDOdbiorcy := sIdAplikacji ,
							sDaneZapasowe := sDaneZapasowe ,
							sDane := sDane ,
							arTablicaKomunikatow := arTablicaKomunikatow ,
							intTablicaKomunikatowZnacznikZapisu := intTablicaKomunikatowZnacznikZapisu ,
							intTablicaKomunikatowRozmiar := intTablicaKomunikatowRozmiar ,
							sWyslanyKomunikat := sWyslanyKomunikat);
	END_IF
END_IF

// Sprawdzanie czy pomiar temperatury działa (odczyt jest niepoprawny, jeśli nie zmienił wartości w przeciągu doby)
IF rTemperaturaPomieszczeniaPamiec = rTemperaturaPomieszczenia THEN
	xBrakZmianyTemperatury := TRUE;
ELSE
	xBrakZmianyTemperatury := FALSE;	
END_IF
fbBrakZmianyTemperaturyTimer(IN := xBrakZmianyTemperatury, PT := T#12H);
rTemperaturaPomieszczeniaPamiec := rTemperaturaPomieszczenia;
IF fbBrakZmianyTemperaturyTimer.Q AND NOT xBrakKomunikacjiPLC THEN
	xBladBrakZmianyTemperatury := TRUE;
ELSE
	xBladBrakZmianyTemperatury := FALSE;
END_IF

// Sprawdzanie czy została osiągnęta zadana temperatura
IF rTemperaturaPomieszczenia >= rTemperaturaNastawiona THEN
	xOsiagniecieTemperaturyZadanej  := TRUE;
END_IF
IF rTemperaturaPomieszczenia <= rTemperaturaNastawiona - 0.4 THEN
	xOsiagniecieTemperaturyZadanej := FALSE;	
END_IF

// obsługa alarmów do zadajnika
	//brak komunikacji po EnOcean
IF arErrorStan[enumPPPSZadajnikError.BrakKomunikacji] <> enumAlarmWartosc.StanAlarmowy AND fbTimeoutEnOcean.Q AND arModbusStatusKomunikacji[bAdres] = enumModbusStatus.KomunikacjaPrawidlowa THEN
	arErrorStan[enumPPPSZadajnikError.BrakKomunikacji] := enumAlarmWartosc.StanAlarmowy;
	xBrakKomunikacjiEnOcean := TRUE;
	arErrorKlasa[enumPPPSZadajnikError.BrakKomunikacji] := enumPPPSZadajnikErrorKlasa.BrakKomunikacji;
	IF xPoInicjalizacji THEN
		fnZapiszKomunikat(	sCalyKomunikat := '' ,
							sTypKomunikatu := 'E' ,
							sMnemonik := sMnemonik ,
							sMACAdres := sMACAdres ,
							sIDNadawcy := sIdInstancji ,
							sIDOdbiorcy := sIdAplikacji ,
							sDaneZapasowe := sDaneZapasowe ,
							sDane := fnKomunikatDaneError(xAktywny := TRUE , intKlasa := enumPPPSZadajnikErrorKlasa.BrakKomunikacji , intNumer := enumPPPSZadajnikError.BrakKomunikacji),
							arTablicaKomunikatow := arTablicaKomunikatow ,
							intTablicaKomunikatowZnacznikZapisu := intTablicaKomunikatowZnacznikZapisu ,
							intTablicaKomunikatowRozmiar := intTablicaKomunikatowRozmiar ,
							sWyslanyKomunikat := sWyslanyKomunikatDummy);
	END_IF
END_IF
IF arErrorStan[enumPPPSZadajnikError.BrakKomunikacji] <> enumAlarmWartosc.StanNormalny AND NOT fbTimeoutEnOcean.Q AND arModbusStatusKomunikacji[bAdres] = enumModbusStatus.KomunikacjaPrawidlowa THEN
	arErrorStan[enumPPPSZadajnikError.BrakKomunikacji] := enumAlarmWartosc.StanNormalny;
	xBrakKomunikacjiEnOcean := FALSE;
	arErrorKlasa[enumPPPSZadajnikError.BrakKomunikacji] := enumPPPSZadajnikErrorKlasa.BrakKomunikacji;
	IF xPoInicjalizacji THEN
		fnZapiszKomunikat(	sCalyKomunikat := '' ,
							sTypKomunikatu := 'E' ,
							sMnemonik := sMnemonik ,
							sMACAdres := sMACAdres ,
							sIDNadawcy := sIdInstancji ,
							sIDOdbiorcy := sIdAplikacji ,
							sDaneZapasowe := sDaneZapasowe ,
							sDane := fnKomunikatDaneError(xAktywny := FALSE , intKlasa := enumPPPSZadajnikErrorKlasa.BrakKomunikacji , intNumer := enumPPPSZadajnikError.BrakKomunikacji),
							arTablicaKomunikatow := arTablicaKomunikatow ,
							intTablicaKomunikatowZnacznikZapisu := intTablicaKomunikatowZnacznikZapisu ,
							intTablicaKomunikatowRozmiar := intTablicaKomunikatowRozmiar ,
							sWyslanyKomunikat := sWyslanyKomunikatDummy);
	END_IF
END_IF
// Alarm czujnika temperatury
IF arErrorStan[enumPPPSZadajnikError.AlarmCzujnika] <> enumAlarmWartosc.StanAlarmowy AND xBladBrakZmianyTemperatury AND arModbusStatusKomunikacji[bAdres] = enumModbusStatus.KomunikacjaPrawidlowa THEN
	arErrorStan[enumPPPSZadajnikError.AlarmCzujnika] := enumAlarmWartosc.StanAlarmowy;
	arErrorKlasa[enumPPPSZadajnikError.AlarmCzujnika] := enumPPPSZadajnikErrorKlasa.AlarmCzujnika;
	IF xPoInicjalizacji THEN
		fnZapiszKomunikat(	sCalyKomunikat := '' ,
							sTypKomunikatu := 'E' ,
							sMnemonik := sMnemonik ,
							sMACAdres := sMACAdres ,
							sIDNadawcy := sIdInstancji ,
							sIDOdbiorcy := sIdAplikacji ,
							sDaneZapasowe := sDaneZapasowe ,
							sDane := fnKomunikatDaneError(xAktywny := TRUE , intKlasa := enumPPPSZadajnikErrorKlasa.AlarmCzujnika , intNumer := enumPPPSZadajnikError.AlarmCzujnika),
							arTablicaKomunikatow := arTablicaKomunikatow ,
							intTablicaKomunikatowZnacznikZapisu := intTablicaKomunikatowZnacznikZapisu ,
							intTablicaKomunikatowRozmiar := intTablicaKomunikatowRozmiar ,
							sWyslanyKomunikat := sWyslanyKomunikatDummy);
	END_IF
END_IF

IF arErrorStan[enumPPPSZadajnikError.AlarmCzujnika] <> enumAlarmWartosc.StanNormalny AND NOT xBladBrakZmianyTemperatury AND arModbusStatusKomunikacji[bAdres] = enumModbusStatus.KomunikacjaPrawidlowa THEN
	arErrorStan[enumPPPSZadajnikError.AlarmCzujnika] := enumAlarmWartosc.StanNormalny;
	arErrorKlasa[enumPPPSZadajnikError.AlarmCzujnika] := enumPPPSZadajnikErrorKlasa.AlarmCzujnika;
	IF xPoInicjalizacji THEN
		fnZapiszKomunikat(	sCalyKomunikat := '' ,
							sTypKomunikatu := 'E' ,
							sMnemonik := sMnemonik ,
							sMACAdres := sMACAdres ,
							sIDNadawcy := sIdInstancji ,
							sIDOdbiorcy := sIdAplikacji ,
							sDaneZapasowe := sDaneZapasowe ,
							sDane := fnKomunikatDaneError(xAktywny := FALSE , intKlasa := enumPPPSZadajnikErrorKlasa.AlarmCzujnika , intNumer := enumPPPSZadajnikError.AlarmCzujnika),
							arTablicaKomunikatow := arTablicaKomunikatow ,
							intTablicaKomunikatowZnacznikZapisu := intTablicaKomunikatowZnacznikZapisu ,
							intTablicaKomunikatowRozmiar := intTablicaKomunikatowRozmiar ,
							sWyslanyKomunikat := sWyslanyKomunikatDummy);
	END_IF
END_IF

// Plakietka pomieszczenia (numer piętra.numer pomieszczenia)
sPlakietkaHMI := CONCAT(STR1 := MID(sIdInstancji, LEN := 2, POS := 3), '.');
sPlakietkaHMI := CONCAT(sPlakietkaHMI, MID(STR := sIdInstancji, LEN := 3, POS := 7));
          
END_FUNCTION_BLOCK

FUNCTION_BLOCK fbTimer
  VAR_INPUT
    xWejscie : BOOL;
    tCzas : TIME;
    tCzasOn : TIME;
    tCzasOff : TIME;
    xReset : BOOL;
    intTyp : INT;
  END_VAR
  VAR_OUTPUT
    xWyjscie : BOOL;
    xError : BOOL;
  END_VAR
  VAR
    negZboczeOpadajace : F_TRIG;
    tCzasowka1 : TON;
    tCzasowka2 : TON;
    xCzasowka1Wyzwolona : BOOL;
    xCzasowka2Wyzwolona : BOOL;
    xCzasowkaStartup : BOOL := TRUE;
  END_VAR

            // Funkcja rozszerzająca funkcjonalność timera

// intTyp - 1 - Opóźnienie włączenia

// xWejscie - sygnał wejściowy zostanie opóźniony na wyjściu xWyjscie po czasie tCzas
// xReset - resetuje czasówkę wznowienie liczenia czasu po powrocie xReset do FALSE
// tCzas - Czas opóźnienia
// tCzasOn - Czas aktywnego wyjścia T#0s - nieskończoność

// intTyp = 2 - Pulse generator

// xWejscie - aktywuje działanie bloku
// tCzasOn - ile czasu xWyjscie ma byc TRUE - jeśli czas = T#0s stan TRUE pojawia się na jeden skan programu
// tCzasOff - ile czasu xWyjscie ma byc FALSE - jeśli czas = T#0s stan FALSE pojawia się na jeden skan programu

// intTyp = 3 - Pulse
// xWejscie - po pojawieniu się xWejscie przez czas tCzas XWyjscie będzie aktywne

// intTyp = 4 -delayed off
// xWejscie aktywne - xWyjscie aktywne, xWejscie deaktywacja - xWyjscie deaktywacja po tCzas

CASE intTyp OF

	1: 
	tCzasowka1(IN:=xWejscie AND NOT xReset,PT:=tCzas);
	IF tCzasOn = T#0S THEN
		xWyjscie := tCzasowka1.Q;
		ELSE
		tCzasowka2(IN := tCzasowka1.Q , PT := tCzasOn);
		xWyjscie := tCzasowka1.Q AND NOT tCzasowka2.Q;
	END_IF

	2:
	tCzasowka1(IN :=  xWejscie AND NOT tCzasowka2.Q , PT := tCzasOff);
	tCzasowka2(IN :=  xWejscie AND tCzasowka1.Q , PT := tCzasOn);
	xWyjscie := tCzasowka1.Q;
		
	3:
	negZboczeOpadajace(CLK := xWejscie);
	tCzasowka1(IN:= xWejscie OR negZboczeOpadajace.Q , PT := tCzas);
	xWyjscie := (xWejscie OR negZboczeOpadajace.Q) AND NOT tCzasowka1.Q;
	
	4:
	negZboczeOpadajace(CLK := xWejscie);
	IF negZboczeOpadajace.Q THEN
		xCzasowkaStartup := FALSE;
	END_IF
	tCzasowka1(IN := NOT negZboczeOpadajace.Q , PT := tCzas);
	xWyjscie := xWejscie OR (NOT tCzasowka1.Q AND NOT xCzasowkaStartup);
	ELSE
		xError := TRUE;
END_CASE;
          
END_FUNCTION_BLOCK

FUNCTION_BLOCK fbUDPComm
  VAR_INPUT
    sIDSterownika : STRING;  (* ID sterownika *)
    sIDAplikacji : STRING;  (* ID aplikacji *)
    sMnemonik : STRING;  (* mnemonik właściciela *)
    sMACAdres : STRING;  (* MAC adres urządzenia - alias *)
    sMACAdresAplikacji : STRING;  (* MAC adres aplikacji - alias *)
    abMACAdresAplikacji : ARRAY[1..6] OF BYTE;  (* MAC adres aplikacji - wartość rzeczywista *)
    sDaneZapasowe : STRING;  (* dane zapasowe *)
    sAdresIP : STRING;  (* adres IP aplikacji *)
    wTransmitterPort : WORD;  (* port do wysyłania komunikatów *)
    wReceiverPort : WORD;  (* port nasłuchu *)
    sKluczSzyfrowania : STRING;
    intTablicaKomunikatowRozmiar : INT;
    intTablicaKomunikatowOverflow : INT;
    intTablicaKomunikatowZnacznikOdczytu : INT;
    iDetekcjaBlokadaKomunikacjiLimitIlosciRamek : INT;  (* Limit ilosi ramek do wysłania *)
    tDetekcjaBlokadaKomunikacjiLimitCzasu : TIME;
  END_VAR
  VAR_IN_OUT
    arTablicaKomunikatow : alARRAYTablicaKomunikatow;
    intTablicaKomunikatowZnacznikZapisu : INT;
    intTablicaKomunikatowZnacznikWysylkiUDP : INT;
    intTablicaKomunikatowLiczbaWBuforze : INT;
    intTransmitterLicznikKomunikatowWyslanych : INT;  (* zmienna zwierająca licznik komunikatów wysłanych pomiędzy heartbetami *)
    intReceiverLicznikKomunikatowOtrzymanych : INT;  (* zmienna zwierająca licznik komunikatów otrzymanych pomiędzy heartbetami *)
  END_VAR
  VAR
    fbTransmitter : fbBroadcaster;  (* definicja drivera wysyłającego broadcast pakietów UDP *)
    udiTransmitterNBytes : UDINT;  (* parametr drivera - ilość bajtów do wysłania *)
    xTransmitterClose : BOOL;  (* parametr drivera - zamknięcie portu komunikacyjnego *)
    xTransmitterTrigger : BOOL;  (* parametr drivera - uruchomienie wysłania telegramu *)
    sTransmitterTelegram : alSTRINGKomunikat;  (* zmienna zawierająca telegram do wysłania *)
    arTransmitterBuffer : ARRAY[1..512] OF BYTE;  (* tablica WORD bufora wysyłkowego *)
    pTransmitterBuffer : POINTER TO BYTE := ADR(arTransmitterBuffer[1]);  (* parametr drivera - pointer do tablicy bufora dla drivera wysyłającego *)
    fbReceiver : fbUdpReceiver;  (* definicja drivera odbierającego pakiety UDP *)
    xReceiverEnable : BOOL := TRUE;  (* parametr drivera - aktywacja działania drivera *)
    xReceiverOpen : BOOL := TRUE;  (* parametr drivera - otworzenie portu komunikacyjnego *)
    sReceiverTelegram : alSTRINGKomunikat;  (* zmienna zawierająca odebrany telegram *)
    arReceiverBuffer : ARRAY[1..512] OF BYTE;
    pReceiverBuffer : POINTER TO BYTE := ADR(arReceiverBuffer[1]);  (* parametr drivera - pointer do tablicy bufora dla drivera odbierającego *)
    intPetla : INT;  (* zmienna tymczasowa używana dla pętli *)
    arwHeartbeatTelegram : ARRAY[1..512] OF WORD;
    negUdpCommTxDone : F_TRIG;
    wCRC16_standard : WORD;
    intBlad : INT;
    sDane : alSTRINGKomunikat;
    sWyslanyKomunikat : alSTRINGKomunikat;
    typKomunikat : typKomunikat;
    xCRC16PakietOdebranyPoprawny : BOOL;
    arErrorKomunikat : ARRAY[0..20] OF alSTRINGKomunikat;  (* tablica przechowująca ostatni komunikat alarmu z danego kodu *)
    arErrorStan : ARRAY[1..20] OF BOOL;  (* tablica przechowująca stany alarmowe *)
    intTabelaKomunikatowZnacznikOdczytu : INT := 1;
    intEmergencyStopActiveZaraportowana : INT;
    sWyslanyKomunikatDummy : STRING;
    BlokadaKomunikacjiDetekcjaTriger : RS;  (* Blokada wysylania komunikatów *)
    BlokadaKomunikacjiDetekcjaTimer : TON;
    BlokadaKomunikacjiTriger : RS;
    fbBlokadaKomunikacjiTimer : TON;  (* Timer do cyklicznego wysyłania ramki z errorem blokady wysyłania ramek *)
    xBlokadaKomunikacji : BOOL;  (* Blokada komunikacji *)
    BlokadaKomunikacjiTimeDiff : TIME := TIME#200m0s0ms;
    xWyslijErrorBlokadyKomunikacji : BOOL;  (* Zmienna pomocniczna do fbWyslijErrorBlokadyKomunikacji *)
    fbWyslijErrorBlokadyKomunikacji : F_TRIG;  (* Zbocze opadające xWyslijErrorBlokadyKomunikacji *)
    xBlokadaKomunikacjiReset : BOOL;  (* Reset blokady komunikacji *)
    timestamp : STRING;  (* obsługa debugowania problemów z komunikatami *)
    dtCzasLokalny : DT;
    dtCzasKomunikatu : DT;
    tPrzesuniecie : TIME := TIME#5m0s0ms;
    xPrzekroczony : BOOL := FALSE;
    arTablicaBlednychKomunikatow : alARRAYTablicaKomunikatowDebug;
    uintZnacznikTablicyBlednychKomunikatow : UINT := 1;
    intTablicaKomunikatowZnacznikWysylkiUDP_Pamiec : INT := -1;
  END_VAR

            // jeśli wysyłanie telegramu zakończone OK wyczyść zmienną zawierającą telegram oraz wyzeruj licznik komunikatów wysłanych jeśli TO BYł heartbeat
// 2019-04-01 - JC Dodanie blokady wysylania komunikatów w przypadku przekroczenia limitu
// 2019-04-18 - AWy: Wysyłanie ramki z errorem blokady wysyłania ramek co minutę
// 2019-04-19 - AWy: Poprawienie mechanizmu resetu blokady i usunięcie tBlokadaKomunikacjiOpoznienie
// 2019-04-25 - AWy: Przeniesienie xBlokadaKomunikacjiReset z VAR_INPUT do VAR
// 2019-10-24 - AWy: Zmiana tPrzesuniecie na 300 sekund
IF NOT xTransmitterTrigger AND sTransmitterTelegram <> '' THEN
	IF fnKomunikatTyp(sTransmitterTelegram) = 'H' THEN
		intTransmitterLicznikKomunikatowWyslanych := 0;
	END_IF
	sTransmitterTelegram := '';
END_IF

IF sTransmitterTelegram = '' AND intTablicaKomunikatowZnacznikWysylkiUDP <> intTablicaKomunikatowZnacznikZapisu THEN
	fnTablicaKomunikatowInkrementacja(intWskaznik := intTablicaKomunikatowZnacznikWysylkiUDP , intRozmiarTablicy := intTablicaKomunikatowRozmiar);
	WHILE fnKomunikatMACAdres(arTablicaKomunikatow[intTablicaKomunikatowZnacznikWysylkiUDP]) <> sMACAdres AND intTablicaKomunikatowZnacznikWysylkiUDP <> intTablicaKomunikatowZnacznikZapisu DO
		fnTablicaKomunikatowInkrementacja(intWskaznik := intTablicaKomunikatowZnacznikWysylkiUDP , intRozmiarTablicy := intTablicaKomunikatowRozmiar);
 	END_WHILE
	IF fnKomunikatMACAdres(arTablicaKomunikatow[intTablicaKomunikatowZnacznikWysylkiUDP]) = sMACAdres THEN
		intTransmitterLicznikKomunikatowWyslanych := intTransmitterLicznikKomunikatowWyslanych + 1;
		//////////////////////////////////
		//Walidacja poprawności komunikatu
		//////////////////////////////////
		IF intTablicaKomunikatowZnacznikWysylkiUDP_Pamiec <> intTablicaKomunikatowZnacznikWysylkiUDP THEN
			timestamp := fnKomunikatSprawdzTimeStamp( sKomunikat:= arTablicaKomunikatow[intTablicaKomunikatowZnacznikWysylkiUDP],dtDataCzasWKomunikacie:=dtCzasKomunikatu, dtDataCzasAktualny:=dtCzasLokalny);
			IF(dtCzasKomunikatu + tPrzesuniecie) < dtCzasLokalny THEN
				xPrzekroczony := TRUE;
				arTablicaBlednychKomunikatow[uintZnacznikTablicyBlednychKomunikatow].dtLokalnyCzasSterownika := dtCzasLokalny;
				arTablicaBlednychKomunikatow[uintZnacznikTablicyBlednychKomunikatow].intGlobalnaLiczbaKomunikatowWBuforze := intTablicaKomunikatowLiczbaWBuforze;
				arTablicaBlednychKomunikatow[uintZnacznikTablicyBlednychKomunikatow].intGlobalnyZnacznikOdczytu := intTablicaKomunikatowZnacznikOdczytu;
				arTablicaBlednychKomunikatow[uintZnacznikTablicyBlednychKomunikatow].intGlobalnyZnacznikWysylkiUDP := intTablicaKomunikatowZnacznikWysylkiUDP;
				arTablicaBlednychKomunikatow[uintZnacznikTablicyBlednychKomunikatow].intGlobalnyZnacznikZapisu := intTablicaKomunikatowZnacznikZapisu;
				arTablicaBlednychKomunikatow[uintZnacznikTablicyBlednychKomunikatow].sDane := arTablicaKomunikatow[intTablicaKomunikatowZnacznikWysylkiUDP];
				IF uintZnacznikTablicyBlednychKomunikatow < 99 THEN
					uintZnacznikTablicyBlednychKomunikatow := uintZnacznikTablicyBlednychKomunikatow + 1;
				ELSE
					uintZnacznikTablicyBlednychKomunikatow := 1;
				END_IF
				//skasuj atrybuty
				arTablicaKomunikatow[intTablicaKomunikatowZnacznikWysylkiUDP] := MID(arTablicaKomunikatow[intTablicaKomunikatowZnacznikWysylkiUDP], 82, 1);
				arTablicaKomunikatow[intTablicaKomunikatowZnacznikWysylkiUDP] := CONCAT(arTablicaKomunikatow[intTablicaKomunikatowZnacznikWysylkiUDP], 'BLADRAMKI=2');
			ELSE
				xPrzekroczony := FALSE;
			END_IF
			intTablicaKomunikatowZnacznikWysylkiUDP_Pamiec := intTablicaKomunikatowZnacznikWysylkiUDP;
		END_IF
		//////////////////////////////////
		fnAES256Szyfrowanie(	sKomunikat := arTablicaKomunikatow[intTablicaKomunikatowZnacznikWysylkiUDP] , 
								sKlucz := sKluczSzyfrowania , 
								intError := intBlad , 
								sKomunikatZaszyfrowany := sTransmitterTelegram);
		
		fnCRC16Wysylanie(	sKomunikat :=  sTransmitterTelegram,
							arTransmitterBuffer := arTransmitterBuffer ,
							udiTransmitterNBytes := udiTransmitterNBytes);
		xTransmitterTrigger := TRUE;
	END_IF
END_IF

// driver wysyłający pakiety UDP

// Blokada wysyłania komunikatów - po przekroczeniu iDetekcjaBlokadaKomunikacjiLimitIlosciRamek w czasie tDetekcjaBlokadaKomunikacjiLimitCzasu algorytm zatrzyma wysyłanie ramek, ale nie 
// przestanie zapisywać ich do tablicy. Raz na minutę zostanie wysłana ramka E informująca o blokadzie. Funkcjonalność ma na celu zabezpieczenia systemu przed spamowaniem ramkami jako 
// konsekwencji błędów programistycznych. 

BlokadaKomunikacjiDetekcjaTriger(Set := (intTablicaKomunikatowZnacznikZapisu = (intTablicaKomunikatowRozmiar - iDetekcjaBlokadaKomunikacjiLimitIlosciRamek)),
								 RESET1 := (intTablicaKomunikatowZnacznikZapisu = intTablicaKomunikatowRozmiar)); // Sprawdzenie następuje, gdy znacznik jest w połowie tablicy komunikatów
IF BlokadaKomunikacjiDetekcjaTimer.ET <> T#0MS AND BlokadaKomunikacjiDetekcjaTriger.RESET1 = TRUE AND NOT xBlokadaKomunikacjiReset THEN
	BlokadaKomunikacjiTimeDiff := BlokadaKomunikacjiDetekcjaTimer.ET; 
END_IF

IF xBlokadaKomunikacjiReset THEN
	BlokadaKomunikacjiTimeDiff := T#200M;
END_IF

BlokadaKomunikacjiDetekcjaTimer(IN := BlokadaKomunikacjiDetekcjaTriger.Q1, PT := T#100S);
 
BlokadaKomunikacjiTriger(Set := (BlokadaKomunikacjiTimeDiff < tDetekcjaBlokadaKomunikacjiLimitCzasu), RESET1 := xBlokadaKomunikacjiReset, Q1 => xBlokadaKomunikacji); 

IF NOT(xBlokadaKomunikacji) THEN
	udiTransmitterNBytes := INT_TO_UDINT(LEN(sTransmitterTelegram)) + 2;
	fbTransmitter(	sNetName := sAdresIP ,
					wPort := wTransmitterPort , 
					pTxBuffer := pTransmitterBuffer , 
					udiTxNBytes := udiTransmitterNBytes , 
					xClose := xTransmitterClose , 
					xTxTrigger := xTransmitterTrigger);
END_IF

// driver nasłuchujący pakietów UDP

fbReceiver(	wPort := wReceiverPort , 
			pRxBuffer := pReceiverBuffer , 
			udiRxBufferSize := 512 , 
			xRxEnable := xReceiverEnable , 
			xOpen := xReceiverOpen);

// po otrzymaniu pakietu wykonanie zapisu danych kontroli CRC itd

IF fbReceiver.xPacketReceived = TRUE THEN
	sReceiverTelegram := LEFT(sReceiverTelegram , UDINT_TO_INT(fbReceiver.udiRxNBytes));
	fnAES256Odszyfrowanie(	sKomunikatZaszyfrowany := sReceiverTelegram , 
							sKlucz := sKluczSzyfrowania ,
							intError := intBlad ,
							sKomunikat := sReceiverTelegram);

// sprawdzenie CRC otrzymanego komunikatu

	xCRC16PakietOdebranyPoprawny := fnCRC16Odbieranie(	arReceiverBuffer := arReceiverBuffer ,
														udiRxNBytes := fbReceiver.udiRxNBytes ,
														sMACAdresAplikacji := sMACAdresAplikacji ,
														abMACAdresAplikacji := abMACAdresAplikacji ,
														sKomunikat := sReceiverTelegram);
	IF xCRC16PakietOdebranyPoprawny THEN

// CRC poprawne zapis komunikatu do tablicy komunikatów otrzymanych o nie jest to komunikat z tego sterownika

		intReceiverLicznikKomunikatowOtrzymanych := intReceiverLicznikKomunikatowOtrzymanych + 1;

		IF fnKomunikatMACAdres(sReceiverTelegram) <> sMACAdres THEN
			fnZapiszKomunikat(	sCalyKomunikat := sReceiverTelegram ,
								sTypKomunikatu := '' ,
								sMnemonik := '' ,
								sMACAdres := '' ,
								sIDNadawcy := '' ,
								sIDOdbiorcy := '' ,
								sDaneZapasowe := '' ,
								sDane := '' ,
								arTablicaKomunikatow := arTablicaKomunikatow ,
								intTablicaKomunikatowZnacznikZapisu := intTablicaKomunikatowZnacznikZapisu ,
								intTablicaKomunikatowRozmiar := intTablicaKomunikatowRozmiar ,
								sWyslanyKomunikat := sWyslanyKomunikat);
		END_IF
		
// sprawdzenie statusu błędu jeśli błąd był zaraportowany zaraportowanie poprawnego CRC

		IF arErrorStan[enumSystemErrorKlasa.BladCRCWKomunikacieZIZE] THEN
			arErrorStan[enumSystemErrorKlasa.BladCRCWKomunikacieZIZE] := FALSE;
			sDane := CONCAT('ACT=0;CLASS=' , INT_TO_STRING(enumSystemErrorKlasa.BladCRCWKomunikacieZIZE));
			sDane := CONCAT(sDane , ';NUM=');
			sDane := CONCAT(sDane , INT_TO_STRING(enumSystemError.BladCRCWKomunikacieZIZE));
			sDane := CONCAT(sDane , ';E');
			sDane := CONCAT(sDane , fnKonwersjaINT_STRING(intWartosc := enumSystemError.BladCRCWKomunikacieZIZE , intIloscZnakow := 3));
			sDane := CONCAT(sDane , 'ACT=0');
			fnZapiszKomunikat(	sCalyKomunikat := '' ,
								sTypKomunikatu := 'E' ,
								sMnemonik :=  sMnemonik ,
								sMACAdres := sMACAdres ,
								sIDNadawcy := sIdSterownika ,
								sIDOdbiorcy := sIdAplikacji ,
								sDaneZapasowe := sDaneZapasowe ,
								sDane := sDane ,
								arTablicaKomunikatow := arTablicaKomunikatow ,
								intTablicaKomunikatowZnacznikZapisu := intTablicaKomunikatowZnacznikZapisu ,
								intTablicaKomunikatowRozmiar := intTablicaKomunikatowRozmiar ,
								sWyslanyKomunikat := arErrorKomunikat[enumSystemError.BladCRCWKomunikacieZIZE]);
			END_IF
		ELSE

// jeżeli był błąd w CRC komunikatu i poprzednie komunikaty były bez błędu zaraportuj ten błąd z powrotem do IZE

		IF NOT arErrorStan[enumSystemErrorKlasa.BladCRCWKomunikacieZIZE] THEN
			arErrorStan[enumSystemErrorKlasa.BladCRCWKomunikacieZIZE] := TRUE;
			sDane := CONCAT('ACT=1;CLASS=' , INT_TO_STRING(enumSystemErrorKlasa.BladCRCWKomunikacieZIZE));
			sDane := CONCAT(sDane , ';NUM=');
			sDane := CONCAT(sDane , INT_TO_STRING(enumSystemError.BladCRCWKomunikacieZIZE));	
			sDane := CONCAT(sDane , ';E');
			sDane := CONCAT(sDane , fnKonwersjaINT_STRING(intWartosc := enumSystemError.BladCRCWKomunikacieZIZE , intIloscZnakow := 3));
			sDane := CONCAT(sDane , 'ACT=1');
			fnZapiszKomunikat(	sCalyKomunikat := '' ,
								sTypKomunikatu := 'E' ,
								sMnemonik :=  sMnemonik,
								sMACAdres := sMACAdres ,
								sIDNadawcy := sIdSterownika ,
								sIDOdbiorcy := sIdAplikacji ,
								sDaneZapasowe := sDaneZapasowe ,
								sDane := sDane ,
								arTablicaKomunikatow := arTablicaKomunikatow ,
								intTablicaKomunikatowZnacznikZapisu := intTablicaKomunikatowZnacznikZapisu ,
								intTablicaKomunikatowRozmiar := intTablicaKomunikatowRozmiar ,
								sWyslanyKomunikat := arErrorKomunikat[enumSystemError.BladCRCWKomunikacieZIZE]);
		END_IF
	END_IF
END_IF

// obsługa alarmu przepełnienia bufora komunikatów

intTablicaKomunikatowLiczbaWBuforze := intTablicaKomunikatowZnacznikZapisu - intTablicaKomunikatowZnacznikWysylkiUDP;

IF intTablicaKomunikatowLiczbaWBuforze < 0 THEN
	intTablicaKomunikatowLiczbaWBuforze := intTablicaKomunikatowLiczbaWBuforze + intTablicaKomunikatowRozmiar;
END_IF

IF intTablicaKomunikatowLiczbaWBuforze > intTablicaKomunikatowOverflow AND NOT arErrorStan[enumSystemError.ZaDuzaIloscKomunikatowWBuforze] THEN
	arErrorStan[enumSystemError.ZaDuzaIloscKomunikatowWBuforze] := TRUE;
	sDane := CONCAT('ACT=1;CLASS=' , INT_TO_STRING(enumSystemErrorKlasa.ZaDuzaIloscKomunikatowWBuforze));
	sDane := CONCAT(sDane , ';NUM=');
	sDane := CONCAT(sDane , INT_TO_STRING(enumSystemError.ZaDuzaIloscKomunikatowWBuforze));	
	sDane := CONCAT(sDane , ';E');
	sDane := CONCAT(sDane , fnKonwersjaINT_STRING(intWartosc := enumSystemError.ZaDuzaIloscKomunikatowWBuforze , intIloscZnakow := 3));
	sDane := CONCAT(sDane , 'ACT=1');
	fnZapiszKomunikat(	sCalyKomunikat := '' ,
						sTypKomunikatu := 'E' ,
						sMnemonik :=  sMnemonik ,
						sMACAdres := sMACAdres ,
						sIDNadawcy := sIdSterownika ,
						sIDOdbiorcy := sIdAplikacji ,
						sDaneZapasowe := sDaneZapasowe ,
						sDane := sDane ,
						arTablicaKomunikatow := arTablicaKomunikatow ,
						intTablicaKomunikatowZnacznikZapisu := intTablicaKomunikatowZnacznikZapisu ,
						intTablicaKomunikatowRozmiar := intTablicaKomunikatowRozmiar ,
						sWyslanyKomunikat := arErrorKomunikat[enumSystemError.ZaDuzaIloscKomunikatowWBuforze]);						
END_IF
IF  intTablicaKomunikatowLiczbaWBuforze = 0 AND arErrorStan[enumSystemError.ZaDuzaIloscKomunikatowWBuforze] THEN
	arErrorStan[enumSystemError.ZaDuzaIloscKomunikatowWBuforze] := FALSE;
	sDane := CONCAT('ACT=0;CLASS=' , INT_TO_STRING(enumSystemErrorKlasa.ZaDuzaIloscKomunikatowWBuforze));
	sDane := CONCAT(sDane , ';NUM=');
	sDane := CONCAT(sDane , INT_TO_STRING(enumSystemError.ZaDuzaIloscKomunikatowWBuforze));	
	sDane := CONCAT(sDane , ';E');
	sDane := CONCAT(sDane , fnKonwersjaINT_STRING(intWartosc := enumSystemError.ZaDuzaIloscKomunikatowWBuforze , intIloscZnakow := 3));
	sDane := CONCAT(sDane , 'ACT=0');
	fnZapiszKomunikat(	sCalyKomunikat := '' ,
						sTypKomunikatu := 'E' ,
						sMnemonik :=  sMnemonik,
						sMACAdres := sMACAdres ,
						sIDNadawcy := sIdSterownika ,
						sIDOdbiorcy := sIdAplikacji ,
						sDaneZapasowe := sDaneZapasowe ,
						sDane := sDane ,
						arTablicaKomunikatow := arTablicaKomunikatow ,
						intTablicaKomunikatowZnacznikZapisu := intTablicaKomunikatowZnacznikZapisu ,
						intTablicaKomunikatowRozmiar := intTablicaKomunikatowRozmiar ,
						sWyslanyKomunikat := arErrorKomunikat[enumSystemError.ZaDuzaIloscKomunikatowWBuforze]);
END_IF


// obsługa alarmu - blokada wysyłania komunikatów ze względu na za dużą ilość wysyłanych ramek (wysyłanie ramki co 1 minutę)

IF xBlokadaKomunikacji THEN
	arErrorStan[enumSystemError.BlokadaWysylaniaRamek] := TRUE;
	fbBlokadaKomunikacjiTimer(IN := xWyslijErrorBlokadyKomunikacji, PT := T#1M);
	xWyslijErrorBlokadyKomunikacji := TRUE;
	IF fbBlokadaKomunikacjiTimer.Q  THEN														// Wyślij error zaraz co 1 minutę
		xWyslijErrorBlokadyKomunikacji := FALSE;
		intTablicaKomunikatowZnacznikWysylkiUDP := intTablicaKomunikatowZnacznikZapisu;			// Ustaw znacznik wysyłania na aktualnie zapisywanej ramce
		// Sklejenie ramki z komunikatem o błędzie
		sDane := CONCAT('ACT=1;CLASS=' , INT_TO_STRING(enumSystemErrorKlasa.BlokadaWysylaniaRamek));
		sDane := CONCAT(sDane , ';NUM=');
		sDane := CONCAT(sDane , INT_TO_STRING(enumSystemError.BlokadaWysylaniaRamek));	
		sDane := CONCAT(sDane , ';E');
		sDane := CONCAT(sDane , fnKonwersjaINT_STRING(intWartosc := enumSystemError.BlokadaWysylaniaRamek , intIloscZnakow := 3));
		sDane := CONCAT(sDane , 'ACT=1');
		fnZapiszKomunikat(	sCalyKomunikat := '' ,
							sTypKomunikatu := 'E' ,
							sMnemonik :=  sMnemonik ,
							sMACAdres := sMACAdres ,
							sIDNadawcy := sIdSterownika ,
							sIDOdbiorcy := sIdAplikacji ,
							sDaneZapasowe := sDaneZapasowe ,
							sDane := sDane ,
							arTablicaKomunikatow := arTablicaKomunikatow ,
							intTablicaKomunikatowZnacznikZapisu := intTablicaKomunikatowZnacznikZapisu ,
							intTablicaKomunikatowRozmiar := intTablicaKomunikatowRozmiar ,
							sWyslanyKomunikat := arErrorKomunikat[enumSystemError.BlokadaWysylaniaRamek]);
		sTransmitterTelegram := arErrorKomunikat[enumSystemError.BlokadaWysylaniaRamek];	
	END_IF
	fbWyslijErrorBlokadyKomunikacji(CLK := xWyslijErrorBlokadyKomunikacji);
	IF fbWyslijErrorBlokadyKomunikacji.Q THEN
		// Wysłanie ramki		
		fnCRC16Wysylanie(	sKomunikat :=  sTransmitterTelegram,
							arTransmitterBuffer := arTransmitterBuffer ,
							udiTransmitterNBytes := udiTransmitterNBytes);				
		udiTransmitterNBytes := INT_TO_UDINT(LEN(sTransmitterTelegram)) + 2;
		fbTransmitter(	sNetName := sAdresIP ,
						wPort := wTransmitterPort , 
						pTxBuffer := pTransmitterBuffer , 
						udiTxNBytes := udiTransmitterNBytes , 
						xClose := xTransmitterClose , 
						xTxTrigger := xTransmitterTrigger);
	END_IF
END_IF
IF  NOT (BlokadaKomunikacjiTriger.Q1) AND arErrorStan[enumSystemError.BlokadaWysylaniaRamek] THEN
	arErrorStan[enumSystemError.BlokadaWysylaniaRamek] := FALSE;
	sDane := CONCAT('ACT=0;CLASS=' , INT_TO_STRING(enumSystemErrorKlasa.BlokadaWysylaniaRamek));
	sDane := CONCAT(sDane , ';NUM=');
	sDane := CONCAT(sDane , INT_TO_STRING(enumSystemError.BlokadaWysylaniaRamek));	
	sDane := CONCAT(sDane , ';E');
	sDane := CONCAT(sDane , fnKonwersjaINT_STRING(intWartosc := enumSystemError.BlokadaWysylaniaRamek , intIloscZnakow := 3));
	sDane := CONCAT(sDane , 'ACT=0');
	fnZapiszKomunikat(	sCalyKomunikat := '' ,
						sTypKomunikatu := 'E' ,
						sMnemonik :=  sMnemonik,
						sMACAdres := sMACAdres ,
						sIDNadawcy := sIdSterownika ,
						sIDOdbiorcy := sIdAplikacji ,
						sDaneZapasowe := sDaneZapasowe ,
						sDane := sDane ,
						arTablicaKomunikatow := arTablicaKomunikatow ,
						intTablicaKomunikatowZnacznikZapisu := intTablicaKomunikatowZnacznikZapisu ,
						intTablicaKomunikatowRozmiar := intTablicaKomunikatowRozmiar ,
						sWyslanyKomunikat := arErrorKomunikat[enumSystemError.BlokadaWysylaniaRamek]);
END_IF


//????????
IF intTabelaKomunikatowZnacznikOdczytu <> intTablicaKomunikatowZnacznikZapisu THEN
	fnTablicaKomunikatowInkrementacja(intRozmiarTablicy := intTablicaKomunikatowRozmiar , intWskaznik := intTabelaKomunikatowZnacznikOdczytu);
	IF fnIDOdbiorcyMatch(arTablicaKomunikatow[intTabelaKomunikatowZnacznikOdczytu] , sIDSterownika) THEN
		IF fnKomunikatTyp(arTablicaKomunikatow[intTabelaKomunikatowZnacznikOdczytu]) = 'Q' THEN
//			IF fnKomunikatDaneSzukajZmiennej(arTablicaKomunikatow[intTabelaKomunikatowZnacznikOdczytu] , 'ALARM') OR 
//				fnKomunikatDaneSzukajZmiennej(arTablicaKomunikatow[intTabelaKomunikatowZnacznikOdczytu] , 'ALL') THEN
//				FOR intPetla := 1 TO 20 BY 1 DO
//					IF arErrorKomunikat[intPetla] <> '' THEN
//						fnZapiszKomunikat(	sCalyKomunikat := arErrorKomunikat[intPetla] ,
//											sTypKomunikatu := '' ,
//											sMnemonik := '' ,
//											sMACAdres := '' ,
//											sIDNadawcy := '' ,
//											sIDOdbiorcy := '' ,
//											sDaneZapasowe := '' ,
//											sDane := '' ,
//											arTablicaKomunikatow := arTablicaKomunikatow ,
//											intTablicaKomunikatowZnacznikZapisu := intTablicaKomunikatowZnacznikZapisu ,
//											intTablicaKomunikatowRozmiar := intTablicaKomunikatowRozmiar ,
//											sWyslanyKomunikat := sWyslanyKomunikat);
//					END_IF
//				END_FOR
//			END_IF	
///wrzucic nowy Q
		END_IF
	END_IF
END_IF
          
END_FUNCTION_BLOCK

FUNCTION fnAES256Odszyfrowanie : BOOL
  VAR_INPUT
    sKomunikatZaszyfrowany : alSTRINGKomunikat;
    sKlucz : STRING;
  END_VAR
  VAR_IN_OUT
    intError : INT;
    sKomunikat : alSTRINGKomunikat;
  END_VAR

            sKomunikat := sKomunikatZaszyfrowany;
          
END_FUNCTION

FUNCTION fnAES256Szyfrowanie : BOOL
  VAR_INPUT
    sKomunikat : alSTRINGKomunikat;
    sKlucz : STRING;
  END_VAR
  VAR_IN_OUT
    intError : INT;
    sKomunikatZaszyfrowany : alSTRINGKomunikat;
  END_VAR

            sKomunikatZaszyfrowany := sKomunikat;
          
END_FUNCTION

FUNCTION fnCRC16Obliczanie : WORD
  VAR_INPUT
    sKomunikat : alSTRINGKomunikat;
  END_VAR
  VAR
    intPetla : INT;
    wCRC16_modbus : WORD;
    arTransmitterBuffer : ARRAY[1..512] OF BYTE;
  END_VAR

            FOR intPetla := 1 TO LEN(sKomunikat) BY 1 DO
	arTransmitterBuffer[intPetla] := string_to_ASCIIByte(MID(sKomunikat , 1 , intPetla));
END_FOR

fnCRC16Obliczanie := MEM.CRC16_modbus(ADR(arTransmitterBuffer[1]) , INT_TO_UINT(LEN(sKomunikat)));
          
END_FUNCTION

FUNCTION fnCRC16Odbieranie : BOOL
  VAR_INPUT
    arReceiverBuffer : ARRAY[1..512] OF BYTE;
    udiRxNBytes : UDINT;
    sMACAdresAplikacji : STRING;
    abMACAdresAplikacji : ARRAY[1..6] OF BYTE;
  END_VAR
  VAR_IN_OUT
    sKomunikat : alSTRINGKomunikat;
  END_VAR
  VAR
    wCRC16_modbus : WORD;
    intPetla : INT;
    arwTelegram : ARRAY[1..512] OF BYTE;
  END_VAR

            wCRC16_modbus := MEM.CRC16_modbus(ADR(arReceiverBuffer[1]) , UDINT_TO_UINT(udiRxNBytes) - 2);
sKomunikat := '';
IF (MEM.LowByte(wCRC16_modbus) = arReceiverBuffer[udiRxNBytes - 1] AND MEM.HighByte(wCRC16_modbus) = arReceiverBuffer[udiRxNBytes]) OR ASCIIByte_to_string(arReceiverBuffer[1]) = 'Z' THEN
	fnCRC16Odbieranie := TRUE;
	FOR intPetla := 1 TO (UDINT_TO_INT(udiRxNBytes) - 2) BY 1 DO
		IF intPetla >= 7 AND intPetla <= 12 AND arReceiverBuffer[7] = abMACAdresAplikacji[1] AND arReceiverBuffer[8] = abMACAdresAplikacji[2] AND arReceiverBuffer[9] = abMACAdresAplikacji[3] AND 
			arReceiverBuffer[10] = abMACAdresAplikacji[4] AND arReceiverBuffer[11] = abMACAdresAplikacji[5] AND arReceiverBuffer[12] = abMACAdresAplikacji[6] THEN
			sKomunikat := CONCAT(sKomunikat , MID(sMACAdresAplikacji, 1 , intPetla - 6));
		ELSE
			sKomunikat := CONCAT(sKomunikat , ASCIIByte_to_string(arReceiverBuffer[intPetla]));
		END_IF
	END_FOR
	ELSE
	fnCRC16Odbieranie := FALSE;	
END_IF

          
END_FUNCTION

FUNCTION fnCRC16Walidacja : BOOL
  VAR_INPUT
    sKomunikat : alSTRINGKomunikat;
    wCRC16Wynik : WORD;
  END_VAR
  VAR
    wCRC16_modbus : WORD;
    intPetla : INT;
    arwTelegram : ARRAY[1..512] OF BYTE;
  END_VAR

            wCRC16_modbus := fnCRC16Obliczanie(sKomunikat);

IF wCRC16_modbus = wCRC16Wynik THEN
	fnCRC16Walidacja := TRUE;
	ELSE	
	fnCRC16Walidacja := FALSE;
END_IF

          
END_FUNCTION

FUNCTION fnCRC16Wysylanie : WORD
  VAR_INPUT
    sKomunikat : alSTRINGKomunikat;
  END_VAR
  VAR_IN_OUT
    arTransmitterBuffer : ARRAY[1..512] OF BYTE;
    udiTransmitterNBytes : UDINT;
  END_VAR
  VAR
    intPetla : INT;
    wCRC16_modbus : WORD;
  END_VAR

            FOR intPetla := 1 TO LEN(sKomunikat) BY 1 DO
	arTransmitterBuffer[intPetla] := string_to_ASCIIByte(MID(sKomunikat , 1 , intPetla));
END_FOR

wCRC16_modbus := fnCRC16Obliczanie(sKomunikat);

arTransmitterBuffer[LEN(sKomunikat) + 1] := MEM.LowByte(wCRC16_modbus);
arTransmitterBuffer[LEN(sKomunikat) + 2] := MEM.HighByte(wCRC16_modbus);

udiTransmitterNBytes := INT_TO_UDINT(LEN(sKomunikat)) + 2;	

fnCRC16Wysylanie := wCRC16_modbus;
          
END_FUNCTION

(* funkcja bez parametrów zwracająca STRING z bieżącym czasem UTC *)
FUNCTION fnCzasUTC : alSTRINGKomunikat
  VAR
    sCzasUTC : STRING;  (* zmienna do przechowywania wyniku - czas w formacie UTC *)
    dtDataIGodzina : DT;  (* odczyt daty i godziny z systemu *)
    ltGodzina : LTIME;  (* odczyt ms z systemu *)
    sDataiGodzina : STRING;  (* odczyt daty i godziny z systemu - konwersja na STRING *)
    sGodzina : STRING;  (* odczyt ms z systemu - konwersjan a STRING *)
    xMsZapisane : BOOL;  (* flaga informująca czy ms zostały już dopisane *)
  END_VAR

            (*odczyt czasu z systemu i jego konwersja do STRING*)

dtDataIGodzina := FuGetDateAndTime();
ltGodzina := FuGetLongTime();
sDataiGodzina := DT_TO_STRING(dtDataiGodzina);
sGodzina := LTIME_TO_STRING(ltGodzina);

sCzasUTC := MID(sDataIGodzina , 4 , 4);							(*dodanie roku do wyniku*)
sCzasUTC := CONCAT(sCzasUTC , '-');
sCzasUTC := CONCAT(sCzasUTC , MID(sDataIGodzina , 2 , 9));		(*dodanie miesiąca do wyniku*)
sCzasUTC := CONCAT(sCzasUTC , '-');
sCzasUTC := CONCAT(sCzasUTC , MID(sDataIGodzina , 2 , 12));		(*dodanie dnia do wyniku*)
sCzasUTC := CONCAT(sCzasUTC , 'T');
sCzasUTC := CONCAT(sCzasUTC , MID(sDataIGodzina , 2 , 15));		(*dodanie godziny do wyniku*)
sCzasUTC := CONCAT(sCzasUTC , ':');
sCzasUTC := CONCAT(sCzasUTC , MID(sDataIGodzina , 2 , 18));		(*dodanie minuty do wyniku*)
sCzasUTC := CONCAT(sCzasUTC , ':');
sCzasUTC := CONCAT(sCzasUTC , MID(sDataIGodzina , 2 , 21));		(*dodanie sekundy do wyniku*)
sCzasUTC := CONCAT(sCzasUTC , '.');

(*sprawdzenie czy w danych o czasie są milisekundy*)

IF FIND(sGodzina , 'ms') <> 0 THEN 

	xMsZapisane := FALSE;

(*jeżeli przed wykrytym 'ms' dwa znaki wcześniej nie ma liczby dopisz dwa zera i liczbę jednocyfrową przed 'ms'*)
		
	IF STRING_TO_INT(MID(sGodzina , 1 , FIND(sGodzina , 'ms') - 2)) = 0 AND MID(sGodzina , 1 , FIND(sGodzina , 'ms') - 2) <> '0' AND xMsZapisane = FALSE THEN
		sCzasUTC := CONCAT(sCzasUTC , '00');
		sCzasUTC := CONCAT(sCzasUTC , MID(sGodzina , 1 , FIND(sGodzina , 'ms') - 1));
		xMsZapisane := TRUE;
	END_IF

(*jeżeli przed wykrytym 'ms' trzy znaki wcześniej nie ma liczby dopisz jedno zero i liczbę dwujcyfrową przed 'ms'*)
		
	IF STRING_TO_INT(MID(sGodzina , 1 , FIND(sGodzina , 'ms') - 3)) = 0 AND MID(sGodzina , 1 , FIND(sGodzina , 'ms') - 3) <> '0' AND xMsZapisane = FALSE THEN
		sCzasUTC := CONCAT(sCzasUTC , '0');
		sCzasUTC := CONCAT(sCzasUTC , MID(sGodzina , 2 , FIND(sGodzina , 'ms') - 2));
		xMsZapisane := TRUE;	
	END_IF

(*jeżeli przed wykrytym 'ms' cztery znaki wcześniej nie ma liczby dopisz liczbę trzycyfrową cyfrową przed 'ms'*)

	IF STRING_TO_INT(MID(sGodzina , 1 , FIND(sGodzina , 'ms') - 4)) = 0 AND MID(sGodzina , 1 , FIND(sGodzina , 'ms') - 4) <> '0' AND xMsZapisane = FALSE THEN
		sCzasUTC := CONCAT(sCzasUTC , MID(sGodzina , 3 , FIND(sGodzina , 'ms') - 3));			
	END_IF
		
	ELSE

(*jeżeli nie wykryto 'ms' dopisz trzy zera*)

	sCzasUTC := CONCAT(sCzasUTC , '000');

END_IF

sCzasUTC := CONCAT(sCzasUTC , '+00:00');

fnCzasUTC :=sCzasUTC;
          
END_FUNCTION

FUNCTION fnIDNadawcyMatch : BOOL
  VAR_INPUT
    sKomunikat : alSTRINGKomunikat;
    sIDObiektu : STRING;
  END_VAR
  VAR
    intPetla : INT;
    xMatch : BOOL := TRUE;
    intBlad : INT;
    typKomunikat : typKomunikat;
  END_VAR

            fnKomunikatInOut(	xStringNaStrukture := TRUE ,
					xStringUpdateZeStruktury := FALSE ,
					xStrukturyNaString := FALSE ,
					xWyczyscStrukture := FALSE ,
					xAktualizujZnacznikCzasu := FALSE ,
					xAktualizujDlugoscDanych := FALSE ,
					sKomunikat := sKomunikat ,
					typKomunikat := typKomunikat ,
					intBlad := intBlad);

FOR intPetla := 1 TO LEN(sIDObiektu) BY 1 DO
	IF (MID(typKomunikat.sIDZrodla , 1 , intPetla) <> MID(sIDObiektu , 1 , intPetla)) AND MID(typKomunikat.sIDZrodla , 1 , intPetla) <> '*' THEN
		xMatch := FALSE;
		EXIT;
	END_IF
END_FOR
fnIDNadawcyMatch := xMatch;
          
END_FUNCTION

FUNCTION fnIDOdbiorcyMatch : BOOL
  VAR_INPUT
    sKomunikat : alSTRINGKomunikat;
    sIDObiektu : STRING;
  END_VAR
  VAR
    typKomunikat : typKomunikat;
    intPetla : INT;
    xMatch : BOOL := TRUE;
    intBlad : INT;
  END_VAR

            fnKomunikatInOut(	xStringNaStrukture := TRUE ,
					xStringUpdateZeStruktury := FALSE ,
					xStrukturyNaString := FALSE ,
					xWyczyscStrukture := FALSE ,
					xAktualizujZnacznikCzasu := FALSE ,
					xAktualizujDlugoscDanych := FALSE ,
					sKomunikat := sKomunikat ,
					typKomunikat := typKomunikat ,
					intBlad := intBlad);

FOR intPetla := 1 TO LEN(sIDObiektu) BY 1 DO
	IF (MID(typKomunikat.sIDPrzeznaczenia , 1 , intPetla) <> MID(sIDObiektu,1,intPetla)) AND MID(typKomunikat.sIDPrzeznaczenia , 1 , intPetla) <> '*' THEN
		xMatch := FALSE;
		EXIT;
	END_IF
END_FOR
fnIDOdbiorcyMatch := xMatch;
          
END_FUNCTION

FUNCTION fnKomunikatDane : STRING
  VAR_INPUT
    sKomunikat : alSTRINGKomunikat;
  END_VAR
  VAR
    intBlad : INT;
    typKomunikat : typKomunikat;
  END_VAR

            fnKomunikatInOut(	xStringNaStrukture := TRUE ,
					xStringUpdateZeStruktury := FALSE ,
					xStrukturyNaString := FALSE ,
					xWyczyscStrukture := FALSE ,
					xAktualizujZnacznikCzasu := FALSE ,
					xAktualizujDlugoscDanych := FALSE ,
					sKomunikat := sKomunikat ,
					typKomunikat := typKomunikat ,
					intBlad := intBlad);
fnKomunikatDane := typKomunikat.sDane;

          
END_FUNCTION

FUNCTION fnKomunikatDaneDodaj : STRING
  VAR_INPUT
    sAtrybut : STRING;
    sWartosc : STRING;
  END_VAR
  VAR_IN_OUT
    sDane : alSTRINGKomunikat;
  END_VAR

            IF sDane <> '' THEN
	sDane := CONCAT(sDane , ';');
END_IF
sDane := CONCAT(sDane , sAtrybut);
sDane := CONCAT(sDane , sWartosc);
          
END_FUNCTION

FUNCTION fnKomunikatDaneDodaj_xOverFlow : STRING
  VAR_INPUT
    sAtrybut : STRING;
    sWartosc : STRING;
  END_VAR
  VAR_IN_OUT
    sDane : alSTRINGKomunikat;
    xOverFlow : BOOL;
  END_VAR
  VAR
    intIloscZnakow : INT;
  END_VAR

            IF sDane <> '' THEN
	sDane := CONCAT(sDane , ';');
END_IF

sDane := CONCAT(sDane , sAtrybut);
sDane := CONCAT(sDane , sWartosc);

intIloscZnakow := len(sDane);
IF intIloscZnakow >= 150 THEN
		xOverFlow := TRUE;
	ELSE
		xOverFlow := FALSE;		
END_IF




          
END_FUNCTION

FUNCTION fnKomunikatDaneDoRaportu_REAL : STRING
  VAR_INPUT
    rWartosc : REAL;
    sAtrybut : STRING;
  END_VAR
  VAR_IN_OUT
    rWartoscZaraportowana : REAL;
    sDane : alSTRINGKomunikat;
  END_VAR

            IF rWartosc <> rWartoscZaraportowana THEN
	rWartoscZaraportowana := rWartosc;
	fnKomunikatDaneDodaj(sDane := sDane , sAtrybut := sAtrybut , sWartosc := REAL_TO_STRING(rWartosc));	
END_IF


          
END_FUNCTION

FUNCTION fnKomunikatDaneError : STRING
  VAR_INPUT
    xAktywny : BOOL;
    intKlasa : INT;
    intNumer : INT;
  END_VAR
  VAR
    sDane : alSTRINGKomunikat;
    typKomunikat : typKomunikat;
  END_VAR

            IF xAktywny THEN
	sDane := CONCAT('ACT=1;CLASS=' , INT_TO_STRING(intKlasa));
	ELSE
	sDane := CONCAT('ACT=0;CLASS=' , INT_TO_STRING(intKlasa));	
END_IF
sDane := CONCAT(sDane , ';NUM=');	
sDane := CONCAT(sDane , INT_TO_STRING(intNumer));
sDane := CONCAT(sDane , ';E');
sDane := CONCAT(sDane , fnKonwersjaINT_STRING(intWartosc := intNumer , intIloscZnakow := 3));
IF xAktywny THEN
	sDane := CONCAT(sDane, 'ACT=1');
	ELSE
	sDane := CONCAT(sDane, 'ACT=0');
END_IF
fnKomunikatDaneError := sDane;

          
END_FUNCTION

FUNCTION fnKomunikatDaneErrorRetry : STRING
  VAR_INPUT
    xAktywny : BOOL;
    intKlasa : INT;
    intNumer : INT;
  END_VAR
  VAR
    sDane : alSTRINGKomunikat;
    typKomunikat : typKomunikat;
  END_VAR

            (* funkcja tylko dla reakcji na Q *)

IF xAktywny THEN
	sDane := CONCAT('RETRY=1;ACT=1;CLASS=' , INT_TO_STRING(intKlasa));
	ELSE
	sDane := CONCAT('RETRY=1;ACT=0;CLASS=' , INT_TO_STRING(intKlasa));	
END_IF
sDane := CONCAT(sDane , ';NUM=');	
sDane := CONCAT(sDane , INT_TO_STRING(intNumer));
sDane := CONCAT(sDane , ';E');
sDane := CONCAT(sDane , fnKonwersjaINT_STRING(intWartosc := intNumer , intIloscZnakow := 3));
IF xAktywny THEN
	sDane := CONCAT(sDane, 'ACT=1');
	ELSE
	sDane := CONCAT(sDane, 'ACT=0');
END_IF
fnKomunikatDaneErrorRetry := sDane;

          
END_FUNCTION

FUNCTION fnKomunikatDaneSzukajWartosci : STRING
  VAR_INPUT
    sKomunikat : alSTRINGKomunikat;
    sZmienna : STRING;
  END_VAR
  VAR
    intBlad : INT;
    typKomunikat : typKomunikat;
    intPozycja1 : INT;
    intPozycja2 : INT;
  END_VAR

            fnKomunikatInOut(	xStringNaStrukture := TRUE ,
					xStringUpdateZeStruktury := FALSE ,
					xStrukturyNaString := FALSE ,
					xWyczyscStrukture := FALSE ,
					xAktualizujZnacznikCzasu := FALSE ,
					xAktualizujDlugoscDanych := FALSE ,
					sKomunikat := sKomunikat ,
					typKomunikat := typKomunikat ,
					intBlad := intBlad);

fnKomunikatDaneSzukajWartosci := typKomunikat.sDane;

IF FIND(typKomunikat.sDane , sZmienna) <> 0 THEN
	fnKomunikatDaneSzukajWartosci := RIGHT(typKomunikat.sDane , LEN(typKomunikat.sDane) - LEN(sZmienna) - FIND(typKomunikat.sDane , sZmienna) + 1);
	IF FIND(fnKomunikatDaneSzukajWartosci , ';') <> 0 THEN
		fnKomunikatDaneSzukajWartosci := LEFT(fnKomunikatDaneSzukajWartosci , FIND(fnKomunikatDaneSzukajWartosci , ';') - 1);
	END_IF
	ELSE
	fnKomunikatDaneSzukajWartosci := '';
END_IF			
          
END_FUNCTION

FUNCTION fnKomunikatDaneSzukajZmiennej : BOOL
  VAR_INPUT
    sKomunikat : alSTRINGKomunikat;
    sZmienna : STRING;
  END_VAR
  VAR
    intBlad : INT;
    typKomunikat : typKomunikat;
    intPozycja1 : INT;
    intPozycja2 : INT;
  END_VAR

            fnKomunikatInOut(	xStringNaStrukture := TRUE ,
					xStringUpdateZeStruktury := FALSE ,
					xStrukturyNaString := FALSE ,
					xWyczyscStrukture := FALSE ,
					xAktualizujZnacznikCzasu := FALSE ,
					xAktualizujDlugoscDanych := FALSE ,
					sKomunikat := sKomunikat ,
					typKomunikat := typKomunikat ,
					intBlad := intBlad);

IF FIND(typKomunikat.sDane , sZmienna) <> 0 THEN
	fnKomunikatDaneSzukajZmiennej := TRUE;
	ELSE
	fnKomunikatDaneSzukajZmiennej := FALSE;
END_IF
				
					
					
					
					
					
					
          
END_FUNCTION

FUNCTION fnKomunikatDaneZnajdzPorownajZapisz : BOOL
  VAR_INPUT
    sKomunikat : alSTRINGKomunikat;  (* Ramka z IZE *)
    sAtrybut : STRING;  (* Atrybut do wyszukania w ramce *)
  END_VAR
  VAR_IN_OUT
    rAtrybutWartosc : REAL;  (* Wartość atrybutu w sterowniku *)
    sDane : STRING;  (* Dane do wysłania w ramce *)
  END_VAR
  VAR_OUTPUT
    xAtrybutZapisz : BOOL;  (* Trigger zapisu wartości atrybutu do urządzenia *)
  END_VAR
  VAR
    sAtrybutWartoscRamka : STRING;  (* Wartość atrybutu z ramki *)
    rAtrybutWartoscRamka : REAL;  (* Wartość atrybutu z ramki *)
  END_VAR

            (*			
Autor:					Artur Wyszomirski, 2019-06-04 
Prawa majątkowe: 		Solwena Sp. z o.o., 
Aktualizacje:			
Opis:					Porównanie wartości atrybutu z ramki przychodzącej z IZE z wartością atrybutu zapisaną w sterowniku (urządzeniu). Jeśli wartość jest różna, triggerowana jest zmienna xAtrybutZapisz (zapis wartości do urządzenia).
						W przeciwnym wypadku nazwa atrybutu i jego wartość przpisywane są do sDane (czyli pola danych ramki A, którą sterownik wyśle w odpowiedzi do IZE) 
*)

sAtrybutWartoscRamka := fnKomunikatDaneSzukajWartosci(sKomunikat, sAtrybut);
// Jeśli wartość atrybutu została odnaleziona w ramce.
IF sAtrybutWartoscRamka <> '' THEN
	rAtrybutWartoscRamka := (STRING_TO_REAL(sAtrybutWartoscRamka));
	// Jeśli wartość różni się od dotychczasowej, zapisz ją. W przeciwnym wypadku doklej wartość do ramki A.
	IF rAtrybutWartoscRamka <> rAtrybutWartosc THEN
		rAtrybutWartosc := rAtrybutWartoscRamka;
		xAtrybutZapisz := TRUE;
	ELSE
		IF sDane <> '' THEN
			sDane := CONCAT(sDane , ';');
		END_IF					
		sDane := CONCAT(sDane , sAtrybut);
		sDane := CONCAT(sDane , sAtrybutWartoscRamka);
	END_IF
END_IF

          
END_FUNCTION

FUNCTION fnKomunikatIDNadawcy : STRING
  VAR_INPUT
    sKomunikat : alSTRINGKomunikat;
  END_VAR
  VAR
    typKomunikat : typKomunikat;
    intBlad : INT;
  END_VAR

            fnKomunikatInOut(	xStringNaStrukture := TRUE ,
					xStringUpdateZeStruktury := FALSE ,
					xStrukturyNaString := FALSE ,
					xWyczyscStrukture := FALSE ,
					xAktualizujZnacznikCzasu := FALSE ,
					xAktualizujDlugoscDanych := FALSE ,
					sKomunikat := sKomunikat ,
					typKomunikat := typKomunikat ,
					intBlad := intBlad);

fnKomunikatIDNadawcy := typKomunikat.sIDPrzeznaczenia;

          
END_FUNCTION

FUNCTION fnKomunikatIDOdbiorcy : STRING
  VAR_INPUT
    sKomunikat : alSTRINGKomunikat;
  END_VAR
  VAR
    typKomunikat : typKomunikat;
    intBlad : INT;
  END_VAR

            fnKomunikatInOut(	xStringNaStrukture := TRUE ,
					xStringUpdateZeStruktury := FALSE ,
					xStrukturyNaString := FALSE ,
					xWyczyscStrukture := FALSE ,
					xAktualizujZnacznikCzasu := FALSE ,
					xAktualizujDlugoscDanych := FALSE ,
					sKomunikat := sKomunikat ,
					typKomunikat := typKomunikat ,
					intBlad := intBlad);

fnKomunikatIDOdbiorcy := typKomunikat.sIDPrzeznaczenia;

          
END_FUNCTION

(* funkcja do kompleksowej obróbki komunikatu *)
FUNCTION fnKomunikatInOut : BOOL
  VAR_INPUT
    xStringNaStrukture : BOOL;  (* rozkaz rozbicia pełnego komunikatu na cząstki *)
    xStringUpdateZeStruktury : BOOL;
    xStrukturyNaString : BOOL;
    xWyczyscStrukture : BOOL;
    xAktualizujZnacznikCzasu : BOOL;  (* rozkaz zaktualizowania znacznika czasu - działa we wszystkich konfiguracjach *)
    xAktualizujDlugoscDanych : BOOL;
  END_VAR
  VAR_IN_OUT
    sKomunikat : alSTRINGKomunikat;
    typKomunikat : typKomunikat;
    intBlad : INT;
  END_VAR
  VAR
    sKomunikatTemp : alSTRINGKomunikat;
  END_VAR

            IF xWyczyscStrukture AND xStringNaStrukture THEN
	fnKomunikatInOutZeruj(typKomunikat);
END_IF
IF xStrukturyNaString THEN
	sKomunikat := CONCAT(typKomunikat.sZnacznik , typKomunikat.sTypKomunikatu);
	sKomunikat := CONCAT(sKomunikat , typKomunikat.sMnemonikWlasciciela);
	sKomunikat := CONCAT(sKomunikat , typKomunikat.sMnemonikWlascicielaExt);
	sKomunikat := CONCAT(sKomunikat , typKomunikat.sMACAdres);	
	IF typKomunikat.sIDZrodla = '' THEN
		sKomunikat := CONCAT(sKomunikat , typKomunikat.sIDZrodlaLokalizacja);
		sKomunikat := CONCAT(sKomunikat , typKomunikat.sIDZrodlaUrzadzenie);
		typKomunikat.sIDZrodla := CONCAT(typKomunikat.sIDZrodlaLokalizacja , typKomunikat.sIDZrodlaUrzadzenie);
		ELSE
		sKomunikat := CONCAT(sKomunikat , typKomunikat.sIDZrodla);
	END_IF
	IF typKomunikat.sIDPrzeznaczenia = '' THEN	
		sKomunikat := CONCAT(sKomunikat , typKomunikat.sIDPrzeznaczeniaLokalizacja);
		sKomunikat := CONCAT(sKomunikat , typKomunikat.sIDPrzeznaczeniaUrzadzenie);
		typKomunikat.sIDPrzeznaczenia := CONCAT(typKomunikat.sIDPrzeznaczeniaLokalizacja , typKomunikat.sIDPrzeznaczeniaUrzadzenie);
		ELSE
		sKomunikat := CONCAT(sKomunikat , typKomunikat.sIDPrzeznaczenia);		
	END_IF
	IF typKomunikat.sDlugoscPolaDanych = '' OR xAktualizujDlugoscDanych THEN
		sKomunikat := CONCAT(sKomunikat ,  fnKonwersjaINT_STRING(intWartosc := LEN(typKomunikat.sDane) , intIloscZnakow := 3));
		typKomunikat.sDlugoscPolaDanych := fnKonwersjaINT_STRING(intWartosc := LEN(typKomunikat.sDane) , intIloscZnakow := 3);
		ELSE
		sKomunikat := CONCAT(sKomunikat , typKomunikat.sDlugoscPolaDanych);
	END_IF
	IF typKomunikat.sMarkerCzasowy = '' OR xAktualizujZnacznikCzasu THEN
		sKomunikat := CONCAT(sKomunikat , fnCzasUTC());
		typKomunikat.sMarkerCzasowy := fnCzasUTC();
		ELSE		
		sKomunikat := CONCAT(sKomunikat , typKomunikat.sMarkerCzasowy);
	END_IF
	sKomunikat := CONCAT(sKomunikat , typKomunikat.sRezerwa);
	sKomunikat := CONCAT(sKomunikat , typKomunikat.sDane);
END_IF

IF xStringNaStrukture OR xStringUpdateZeStruktury THEN
	IF typKomunikat.sZnacznik <> '' AND xStringUpdateZeStruktury THEN
		sKomunikat := CONCAT(typKomunikat.sZnacznik , MID(sKomunikat , LEN(sKomunikat) - 1 , 2));
		ELSE
		typKomunikat.sZnacznik := LEFT(sKomunikat , 1);
	END_IF
	IF typKomunikat.sTypKomunikatu <> '' AND xStringUpdateZeStruktury THEN
		sKomunikatTemp := LEFT(sKomunikat , 1);
		sKomunikat := CONCAT(typKomunikat.sTypKomunikatu , MID(sKomunikat , LEN(sKomunikat) - 2 , 3));
		sKomunikat := CONCAT(sKomunikatTemp , sKomunikat);
		ELSE
		typKomunikat.sTypKomunikatu := MID(SKomunikat , 1 , 2);
	END_IF
	IF typKomunikat.sMnemonikWlasciciela <> '' AND xStringUpdateZeStruktury THEN
		sKomunikatTemp := LEFT(sKomunikat , 2);
		sKomunikat := CONCAT(typKomunikat.sMnemonikWlasciciela , MID(sKomunikat , LEN(sKomunikat) - 5 , 6));
		sKomunikat := CONCAT(sKomunikatTemp , sKomunikat);
		ELSE
		typKomunikat.sMnemonikWlasciciela := MID(sKomunikat , 3 , 3);
	END_IF
	IF typKomunikat.sMnemonikWlascicielaExt <> '' AND xStringUpdateZeStruktury THEN
		sKomunikatTemp := LEFT(sKomunikat , 5);
		sKomunikat := CONCAT(typKomunikat.sMnemonikWlascicielaExt , MID(sKomunikat , LEN(sKomunikat) - 6 , 7));
		sKomunikat := CONCAT(sKomunikatTemp , sKomunikat);
		ELSE
		typKomunikat.sMnemonikWlascicielaExt := MID(Skomunikat , 1 , 6);
	END_IF
	IF typKomunikat.sMACAdres <> '' AND xStringUpdateZeStruktury THEN
		sKomunikatTemp := LEFT(sKomunikat , 6);
		sKomunikat := CONCAT(typKomunikat.sMnemonikWlascicielaExt , MID(sKomunikat , LEN(sKomunikat) - 12 , 13));
		sKomunikat := CONCAT(sKomunikatTemp , sKomunikat);
		ELSE
		typKomunikat.sMACAdres := MID(sKomunikat , 6 , 7);
	END_IF
	IF typKomunikat.sIDZrodla <> '' AND xStringUpdateZeStruktury THEN
		sKomunikatTemp := LEFT(sKomunikat , 12);
		sKomunikat := CONCAT(typKomunikat.sIDZrodla , MID(sKomunikat , LEN(sKomunikat) - 28 , 29));
		sKomunikat := CONCAT(sKomunikatTemp , sKomunikat);
		ELSE
		typKomunikat.sIDZrodla := MID(sKomunikat , 16 , 13);
	END_IF
	IF typKomunikat.sIDZrodlaLokalizacja <> '' AND xStringUpdateZeStruktury THEN
		sKomunikatTemp := LEFT(sKomunikat , 12);
		sKomunikat := CONCAT(typKomunikat.sIDZrodlaLokalizacja , MID(sKomunikat , LEN(sKomunikat) - 24 , 25));
		sKomunikat := CONCAT(sKomunikatTemp , sKomunikat);
		ELSE
		typKomunikat.sIDZrodlaLokalizacja := MID(SKomunikat , 12 , 13);
	END_IF
	IF typKomunikat.sIDZrodlaUrzadzenie <> '' AND xStringUpdateZeStruktury THEN
		sKomunikatTemp := LEFT(sKomunikat , 24);
		sKomunikat := CONCAT(typKomunikat.sIDZrodlaUrzadzenie , MID(sKomunikat , LEN(sKomunikat) - 28 , 29));
		sKomunikat := CONCAT(sKomunikatTemp , sKomunikat);
		ELSE
		typKomunikat.sIDZrodlaUrzadzenie := MID(SKomunikat , 4 , 25);		
	END_IF
	IF typKomunikat.sIDPrzeznaczenia <> '' AND xStringUpdateZeStruktury THEN
		sKomunikatTemp := LEFT(sKomunikat , 28);
		sKomunikat := CONCAT(typKomunikat.sIDPrzeznaczenia , MID(sKomunikat , LEN(sKomunikat) - 44 ,45));
		sKomunikat := CONCAT(sKomunikatTemp , sKomunikat);
		ELSE
		typKomunikat.sIDPrzeznaczenia := MID(SKomunikat , 16 , 29);
	END_IF
	IF typKomunikat.sIDPrzeznaczeniaLokalizacja <> '' AND xStringUpdateZeStruktury THEN
		sKomunikatTemp := LEFT(sKomunikat , 28);
		sKomunikat := CONCAT(typKomunikat.sIDPrzeznaczeniaLokalizacja , MID(sKomunikat , LEN(sKomunikat) - 40 ,41));
		sKomunikat := CONCAT(sKomunikatTemp , sKomunikat);
		ELSE
		typKomunikat.sIDPrzeznaczeniaLokalizacja := MID(SKomunikat , 12 , 29);
	END_IF
	IF typKomunikat.sIDPrzeznaczeniaUrzadzenie <> '' AND xStringUpdateZeStruktury THEN
		sKomunikatTemp := LEFT(sKomunikat , 40);
		sKomunikat := CONCAT(typKomunikat.sIDPrzeznaczeniaUrzadzenie , MID(sKomunikat , LEN(sKomunikat) - 44 ,45));
		sKomunikat := CONCAT(sKomunikatTemp , sKomunikat);
		ELSE
		typKomunikat.sIDPrzeznaczeniaUrzadzenie := MID(SKomunikat , 4 , 41);
	END_IF
	IF typKomunikat.sMarkerCzasowy <> '' AND xStringUpdateZeStruktury THEN
		IF xAktualizujZnacznikCzasu THEN
			sKomunikatTemp := LEFT(sKomunikat , 47);
			sKomunikat := CONCAT(fnCzasUTC() , MID(sKomunikat , LEN(sKomunikat) - 76 , 77));			
			sKomunikat := CONCAT(sKomunikatTemp , sKomunikat);
			ELSE
			sKomunikatTemp := LEFT(sKomunikat , 47);
			sKomunikat := CONCAT(typKomunikat.sMarkerCzasowy , MID(sKomunikat , LEN(sKomunikat) - 76 , 77));
			sKomunikat := CONCAT(sKomunikatTemp , sKomunikat);
		END_IF
		ELSE
		typKomunikat.sMarkerCzasowy := MID(SKomunikat , 29 , 48);
	END_IF
	IF typKomunikat.sRezerwa <> '' AND xStringUpdateZeStruktury THEN
		sKomunikatTemp := LEFT(sKomunikat , 76);
		sKomunikat := CONCAT(typKomunikat.sRezerwa , MID(sKomunikat , LEN(sKomunikat) - 82 , 83));
		sKomunikat := CONCAT(sKomunikatTemp , sKomunikat);
		ELSE
		typKomunikat.sRezerwa := MID(SKomunikat , 6 , 77);
	END_IF
	IF typKomunikat.sDane <> '' AND xStringUpdateZeStruktury THEN
		sKomunikatTemp := LEFT(sKomunikat , 82);
		sKomunikat := CONCAT(sKomunikatTemp , typKomunikat.sDane);
		ELSE
		typKomunikat.sDane := RIGHT(sKomunikat ,  LEN(sKomunikat) - 82);
	END_IF
	IF typKomunikat.sDlugoscPolaDanych <> '' AND xStringUpdateZeStruktury THEN
		IF xAktualizujDlugoscDanych THEN
			sKomunikatTemp := LEFT(sKomunikat , 44);
			sKomunikat := CONCAT(fnKonwersjaINT_STRING(intWartosc := LEN(typKomunikat.sDane) , intIloscZnakow := 3) , MID(sKomunikat , LEN(sKomunikat) - 47 , 48));
			sKomunikat := CONCAT(sKomunikatTemp , sKomunikat);
		ELSE
			sKomunikatTemp := LEFT(sKomunikat , 44);
			sKomunikat := CONCAT(typKomunikat.sDlugoscPolaDanych , MID(sKomunikat , LEN(sKomunikat) - 47 , 48));
			sKomunikat := CONCAT(sKomunikatTemp , sKomunikat);
		END_IF
		ELSE
		typKomunikat.sDlugoscPolaDanych := MID(SKomunikat , 3 , 45);
	END_IF
END_IF

          
END_FUNCTION

FUNCTION fnKomunikatInOutZeruj : BOOL
  VAR_IN_OUT
    typKomunikat : typKomunikat;
  END_VAR

            typKomunikat.sZnacznik := '';
typKomunikat.sTypKomunikatu := '';
typKomunikat.sMnemonikWlasciciela := '';
typKomunikat.sMnemonikWlascicielaExt := '';
typKomunikat.sMACAdres := '';
typKomunikat.sIDZrodla := '';
typKomunikat.sIDZrodlaLokalizacja := '';
typKomunikat.sIDZrodlaUrzadzenie := '';
typKomunikat.sIDPrzeznaczenia :='' ;
typKomunikat.sIDPrzeznaczeniaLokalizacja := '';
typKomunikat.sIDPrzeznaczeniaUrzadzenie := '';
typKomunikat.sDlugoscPolaDanych := '';
typKomunikat.sMarkerCzasowy := '';
typKomunikat.sRezerwa := '';
typKomunikat.sDane := '';
          
END_FUNCTION

FUNCTION fnKomunikatMACAdres : STRING
  VAR_INPUT
    sKomunikat : alSTRINGKomunikat;
  END_VAR
  VAR
    typKomunikat : typKomunikat;
    intBlad : INT;
  END_VAR

            fnKomunikatInOut(	xStringNaStrukture := TRUE ,
					xStringUpdateZeStruktury := FALSE ,
					xStrukturyNaString := FALSE ,
					xWyczyscStrukture := FALSE ,
					xAktualizujZnacznikCzasu := FALSE ,
					xAktualizujDlugoscDanych := FALSE ,
					sKomunikat := sKomunikat ,
					typKomunikat := typKomunikat ,
					intBlad := intBlad);

fnKomunikatMACAdres := typKomunikat.sMACAdres;

          
END_FUNCTION

FUNCTION fnKomunikatMACNadpisanie : STRING
  VAR_INPUT
    abMACAdres : ARRAY[1..6] OF BYTE;
  END_VAR
  VAR_IN_OUT
    sKomunikat : alSTRINGKomunikat;
  END_VAR
  VAR
    intBlad : INT;
    typKomunikat : typKomunikat;
  END_VAR

            

          
END_FUNCTION

FUNCTION fnKomunikatSprawdzTimeStamp : STRING
  VAR_INPUT
    sKomunikat : alSTRINGKomunikat;
  END_VAR
  VAR_IN_OUT
    dtDataCzasWKomunikacie : DT;
    dtDataCzasAktualny : DT;
  END_VAR
  VAR
    sKomunikatDoObrobki : alSTRINGKomunikat;
    sString : STRING;
    uintRok : UINT;
    uintMiesiac : UINT;
    uintDzien : UINT;
    uintGodzina : UINT;
    uintMinuta : UINT;
    uintSekunda : UINT;
  END_VAR

            sKomunikatDoObrobki := sKomunikat;

sString := 'DT#'; 
sString := CONCAT(sString, MID(sKomunikatDoObrobki, 10, 48));
sString := CONCAT(sString, '-'); 
sString := CONCAT(sString, MID(sKomunikatDoObrobki, 8, 59)); 
dtDataCzasWKomunikacie := STRING_TO_DT(sString);
dtDataCzasAktualny := FuGetDateAndTime();

fnKomunikatSprawdzTimeStamp := sString;
          
END_FUNCTION

FUNCTION fnKomunikatTyp : STRING
  VAR_INPUT
    sKomunikat : alSTRINGKomunikat;
  END_VAR
  VAR
    typKomunikat : typKomunikat;
    intBlad : INT;
  END_VAR

            fnKomunikatInOut(	xStringNaStrukture := TRUE ,
					xStringUpdateZeStruktury := FALSE ,
					xStrukturyNaString := FALSE ,
					xWyczyscStrukture := FALSE ,
					xAktualizujZnacznikCzasu := FALSE ,
					xAktualizujDlugoscDanych := FALSE ,
					sKomunikat := sKomunikat ,
					typKomunikat := typKomunikat ,
					intBlad := intBlad);

fnKomunikatTyp := typKomunikat.sTypKomunikatu;

          
END_FUNCTION

